ABB RobotStudio station: c.rspag

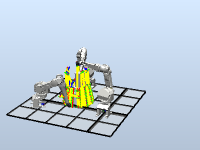
--- station ---
Station c (saved by RobotStudio 6.8.8148.134)
Controller pr3, task T_ROB1: task frame (RAPID world) sits at (2229.65, 1960.18, 0) mm, rotated rx 0 ry 0 rz 180 deg in the station
Controller pr2, task T_ROB1: task frame (RAPID world) sits at (-440.11, 3060.43, 0) mm, rotated rx 0 ry 0 rz -60 deg in the station
Controller pr1
  mechanical unit ROB_1: IRB5510_12A_1100_1500__01, 6 joints, base frame (0, 0, 0) mm
Controller pr2
  mechanical unit ROB_1: IRB5510_12A_1100_1500__01_2, 6 joints, base frame (0, 0, 0) mm
Controller pr3
  mechanical unit ROB_1: IRB5510_12A_1100_1500__01_3, 6 joints, base frame (0, 0, 0) mm
Layout (positions relative to the parent item):
  - IRB5510_12A_1100_1500__01 [mechanism, from Robots\IRB5510_12A_1100_1500__01.rslib] at (0, 0, 0) mm; joint values [1.3542, 0.2117, -0.2881, 5.1047, -1.3259, -6.4536] (rad or m)
  - Workpiece1 [part] at (525.52, 1641.26, 0) mm
  - SmartComponent_1 [smart component]
      signals: DI dipainting
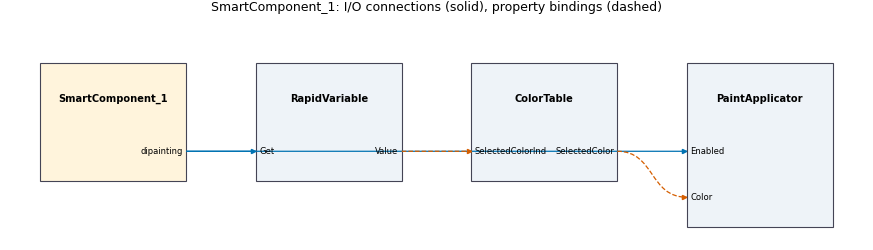
      connections:
        SmartComponent_1.dipainting -> RapidVariable.Get
        SmartComponent_1.dipainting -> PaintApplicator.Enabled
        RapidVariable.Value => ColorTable.SelectedColorIndex
        ColorTable.SelectedColor => PaintApplicator.Color
    - RapidVariable [smart component, from Components\RapidVariable.rslib] at (525.52, 1641.26, 0) mm
        properties: DataType=num; Controller=pr1; Task=T_ROB1; Module=Module1; Variable=ColorIndex; Value=1
    - ColorTable [smart component, from Components\ColorTable.rslib]
        properties: NumColors=2; SelectedColorIndex=1; SelectedColor=-65536; Color0=-8323328; Color1=-65536
    - PaintApplicator [smart component, from Components\PaintApplicator.rslib] at (380.08, 1590.25, 1937.3) mm, rotated rx -165.29 ry -4.8 rz -35.6 deg
        properties: Part=Workpiece1; Color=-65536; ShowPreviewCone=true; Strength=1; Range=0.5; Width=0.1; Height=0.1
  - IRB5510_12A_1100_1500__01_2 [mechanism, from Robots\IRB5510_12A_1100_1500__01.rslib] at (-440.11, 3060.43, 0) mm, rotated rx 0 ry 0 rz -60 deg; joint values [-0.3666, 1.0855, 0.2681, -2.8851, 1.0858, 0.687] (rad or m)
  - SmartComponent_2 [smart component]
      signals: DI dipainting2
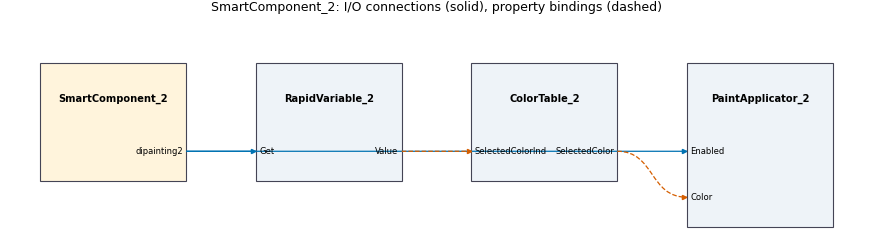
      connections:
        SmartComponent_2.dipainting2 -> RapidVariable_2.Get
        SmartComponent_2.dipainting2 -> PaintApplicator_2.Enabled
        RapidVariable_2.Value => ColorTable_2.SelectedColorIndex
        ColorTable_2.SelectedColor => PaintApplicator_2.Color
    - PaintApplicator_2 [smart component, from Components\PaintApplicator.rslib] at (-112.67, 1718.9, 64) mm, rotated rx -102.66 ry 3.38 rz -125.56 deg
        properties: Part=Workpiece1; Color=-65536; ShowPreviewCone=true; Strength=1; Range=0.5; Width=0.1; Height=0.1
    - RapidVariable_2 [smart component, from Components\RapidVariable.rslib]
        properties: DataType=num; Controller=pr2; Task=T_ROB1; Module=Module1; Variable=ColorIndex2; Value=1
    - ColorTable_2 [smart component, from Components\ColorTable.rslib]
        properties: NumColors=2; SelectedColorIndex=1; SelectedColor=-65536; Color0=-16711936; Color1=-65536
  - IRB5510_12A_1100_1500__01_3 [mechanism, from Robots\IRB5510_12A_1100_1500__01.rslib] at (2229.65, 1960.18, 0) mm, rotated rx 0 ry 0 rz 180 deg; joint values [0.099, 0.1133, 0.783, 6.9211, 0.1129, -9.8516] (rad or m)
  - SmartComponent_3 [smart component]
      signals: DI dipainting3
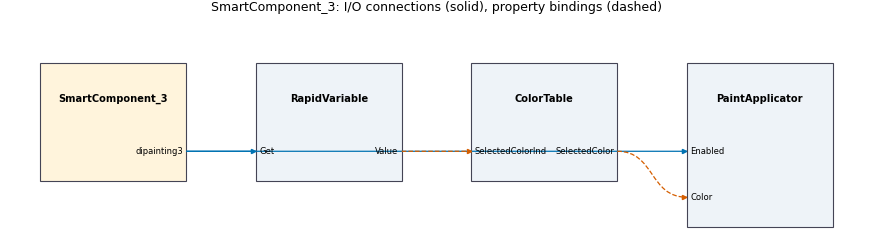
      connections:
        SmartComponent_3.dipainting3 -> RapidVariable.Get
        SmartComponent_3.dipainting3 -> PaintApplicator.Enabled
        RapidVariable.Value => ColorTable.SelectedColorIndex
        ColorTable.SelectedColor => PaintApplicator.Color
    - ColorTable [smart component, from Components\ColorTable.rslib]
        properties: NumColors=2; SelectedColorIndex=1; SelectedColor=-65536; Color0=-16711936; Color1=-65536
    - PaintApplicator [smart component, from Components\PaintApplicator.rslib] at (1182.52, 1870.98, 835.06) mm, rotated rx -177.35 ry -34.28 rz 170.77 deg
        properties: Part=Workpiece1; Color=-65536; ShowPreviewCone=true; Strength=1; Range=0.5; Width=0.1; Height=0.1
    - RapidVariable [smart component, from Components\RapidVariable.rslib]
        properties: DataType=num; Controller=pr3; Task=T_ROB1; Module=Module1; Variable=ColorIndex3; Value=1
Attachment: PaintApplicator is attached to IRB5510_12A_1100_1500__01 / Link6
Attachment: RapidVariable is attached to Workpiece1
Attachment: PaintApplicator_2 is attached to IRB5510_12A_1100_1500__01_2 / Link6
Attachment: PaintApplicator is attached to IRB5510_12A_1100_1500__01_3 / Link6
Station logic (signal -> signal, property => property):
  pr1.do1 -> SmartComponent_1.dipainting
  pr2.do2 -> SmartComponent_2.dipainting2
  pr3.do3 -> SmartComponent_3.dipainting3
Targets, tools, work objects and paths stored in the station and not in the controller backup, written as RAPID:
! task T_ROB1
MODULE Module1
  CONST robtarget Target_20_8_1:=[[1168.457580802,482.978083743,355.510491805],[0.383636594,-0.280466499,0.519275457,-0.710291846],[0,0,0,0],[9E+09,9E+09,9E+09,9E+09,9E+09,9E+09]];
ENDMODULE


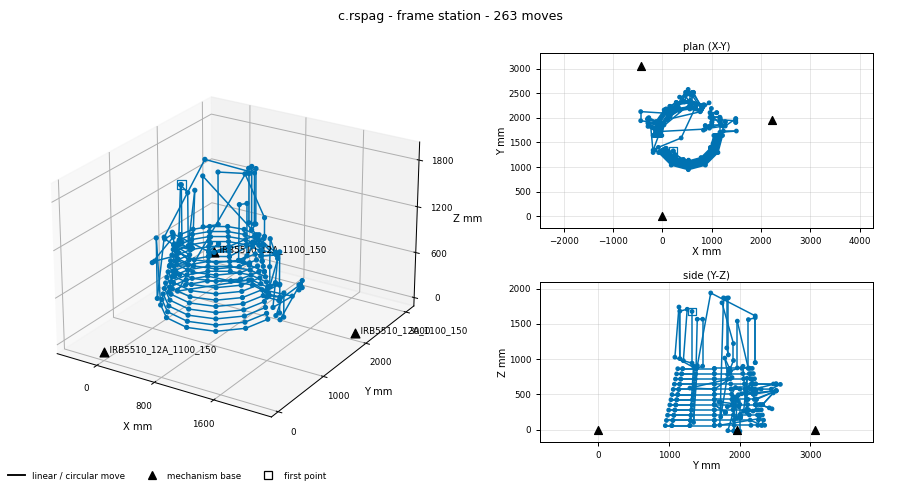
[picture p0: tool path of c.rspag in frame station, 263 of 265 moves have a stored position in this frame; points joined in program order, loops and branches not executed]
--- Backups/pr1/RAPID/TASK0/SYSMOD/userlog.sys ---
module userlog(sysmodule)



   local const num MAX_LOG_SIZE   := 100000; ! Size in bytes.
   local const num MAX_LOG_FILES  := 5;
   local const num MAX_LOG_BUFFER := 20; ! Entries to keep before flushing.



   ! Keep persistent to survive restarts and share between tasks.
   pers string stUserLogBuffer{MAX_LOG_BUFFER};
   pers string stUserLogTime{MAX_LOG_BUFFER};
   pers num nUserLogIndex;
   pers num nUserLogFileNo;

   pers bool bUserBufAddSem;
   pers bool bUserFlushSem;



   proc PntUserLog(string stMessage \Switch Flush)
      BufferAdd stMessage;
      if Present(Flush)
         FlushBuffer;
   endproc



   local proc BufferAdd(string stMessage)
      var bool bTimeOut;

      WaitUntil TestAndSet(bUserBufAddSem) \MaxTime := 1 \TimeFlag := bTimeOut;
      if bTimeOut then
         ErrWrite "PntUserLog Error", "Buffer Add Semaphore Timeout";
         bUserBufAddSem := false; ! Force release.
         return;
      endif

      stUserLogBuffer{nUserLogIndex} := stMessage;
      stUserLogTime{nUserLogIndex} := CDate() + " " + CTime();

      Incr nUserLogIndex;
      if nUserLogIndex > MAX_LOG_BUFFER then
         ! Must be flushed.
         FlushBuffer;
      endif

      bUserBufAddSem := false; ! Release.
   error
      if errno = ERR_OUTOFBND then
         Decr nUserLogIndex;
         retry;
      endif
   endproc



   local proc FlushBuffer()
      var bool bTimeOut;
      var iodev ioLog;
      var string stLogFile;

      WaitUntil TestAndSet(bUserFlushSem) \MaxTime := 1 \TimeFlag := bTimeOut;
      if bTimeOut then
         ErrWrite "PntUserLog Error", "Flush Semaphore Timeout";
         bUserFlushSem := false; ! Force release.
         return;
      endif

      if nUserLogIndex <= 1 then
         bUserFlushSem := false;
         return; ! Buffer empty, nothing to flush.
      endif

      stLogFile := "HOME:/logs/user" + ValToStr(nUserLogFileNo) + ".log";

      Open stLogFile, ioLog \Append;
      for i from 1 to nUserLogIndex - 1 do ! Will normally be incremented to one above.
         Write ioLog, stUserLogTime{i} + " " \NoNewLine;
         Write ioLog, stUserLogBuffer{i};
      endfor
      Close ioLog;
      nUserLogIndex := 1;

      if FileSize(stLogFile) > MAX_LOG_SIZE then
         Incr nUserLogFileNo;
         if nUserLogFileNo > MAX_LOG_FILES
            nUserLogFileNo := 1;

         stLogFile := "HOME:/logs/user" + ValToStr(nUserLogFileNo) + ".log";
         Open stLogFile, ioLog;
         Close ioLog;
      endif

      bUserFlushSem := false;
   error
      nUserLogIndex := 1;
      bUserFlushSem := false;
      return;
   endproc



   proc InitUserLog()
      bUserBufAddSem := false;
      bUserFlushSem := false;
      if nUserLogIndex = 0
         nUserLogIndex := 1;
      if nUserLogFileNo = 0
         nUserLogFileNo := 1;
   endproc



endmodule

--- Backups/pr1/RAPID/TASK1/PROGMOD/Module1.mod ---
MODULE Module1
	CONST robtarget Target_10:=[[220.972076113,1325.461164863,1675.045963445],[0.428514417,-0.848693424,-0.003788423,-0.309968569],[0,-2,0,-1],[9E+09,9E+09,9E+09,9E+09,9E+09,9E+09]];
	CONST robtarget Target_20:=[[220.972027283,1325.461318707,943.383318713],[0.428514341,-0.848693578,-0.003788679,-0.30996825],[0,-3,1,-1],[9E+09,9E+09,9E+09,9E+09,9E+09,9E+09]];
	CONST robtarget Target_30:=[[255.876169889,1202.287029937,977.735293127],[0.428514201,-0.848694161,-0.00378949,-0.309966838],[0,-3,1,-1],[9E+09,9E+09,9E+09,9E+09,9E+09,9E+09]];
	CONST robtarget Target_40:=[[255.876146336,1256.809125064,1706.135963599],[0.428515168,-0.848693816,-0.003790024,-0.30996644],[0,-2,0,-1],[9E+09,9E+09,9E+09,9E+09,9E+09,9E+09]];

    CONST robtarget Target_50:=[[423.854082514,1152.351337183,1679.753004286],[0.470738228,-0.862443821,-0.062003712,-0.175361671],[0,-1,-1,-1],[9E+09,9E+09,9E+09,9E+09,9E+09,9E+09]];
    CONST robtarget Target_60:=[[423.854188981,1152.351291133,1007.412938276],[0.470738104,-0.862443793,-0.062004223,-0.17536196],[0,0,-3,-1],[9E+09,9E+09,9E+09,9E+09,9E+09,9E+09]];
    PERS num ColorIndex:=1;
	CONST robtarget Target_70:=[[530.439659908,1082.627182458,1027.159892696],[0.48639792,-0.862240028,-0.096330933,-0.103341902],[0,0,-2,-1],[9E+09,9E+09,9E+09,9E+09,9E+09,9E+09]];
	CONST robtarget Target_100:=[[76.862753625,1382.222294523,864.109062315],[0.54301355,-0.674637975,0.389502299,-0.313508925],[0,0,0,0],[9E+09,9E+09,9E+09,9E+09,9E+09,9E+09]];
	CONST robtarget Target_110:=[[266.489526282,1192.595596051,864.109062259],[0.605652882,-0.752460843,0.201621223,-0.162284158],[0,0,0,0],[9E+09,9E+09,9E+09,9E+09,9E+09,9E+09]];
	CONST robtarget Target_120:=[[525.524468822,1123.187410427,864.109061963],[0.627017992,-0.779004774,0,0],[0,-2,0,0],[9E+09,9E+09,9E+09,9E+09,9E+09,9E+09]];
	CONST robtarget Target_130:=[[784.559411363,1192.595596051,864.109062259],[0.605652882,-0.752460843,-0.201621223,0.162284158],[0,0,0,0],[9E+09,9E+09,9E+09,9E+09,9E+09,9E+09]];
	CONST robtarget Target_140:=[[974.18618402,1382.222294523,864.109062315],[0.54301355,-0.674637975,-0.389502299,0.313508925],[0,0,0,0],[9E+09,9E+09,9E+09,9E+09,9E+09,9E+09]];
	CONST robtarget Target_150:=[[1043.594471035,1641.25720958,864.109061867],[0.443368761,-0.550839666,-0.55083945,0.443368587],[0,1,1,1],[9E+09,9E+09,9E+09,9E+09,9E+09,9E+09]];
	CONST robtarget Target_150_2:=[[1059.621736679,1641.257203305,790.841560504],[0.443368761,-0.550839666,-0.55083945,0.443368587],[0,1,1,1],[9E+09,9E+09,9E+09,9E+09,9E+09,9E+09]];
	CONST robtarget Target_140_2:=[[988.066201213,1374.208657999,790.841560977],[0.54301355,-0.674637975,-0.389502299,0.313508925],[0,0,0,0],[9E+09,9E+09,9E+09,9E+09,9E+09,9E+09]];
	CONST robtarget Target_130_2:=[[792.573042484,1178.715575754,790.841560918],[0.605652882,-0.752460843,-0.201621223,0.162284158],[0,0,0,0],[9E+09,9E+09,9E+09,9E+09,9E+09,9E+09]];
	CONST robtarget Target_120_2:=[[525.524468822,1107.160144759,790.841560605],[0.627017992,-0.779004774,0,0],[0,-2,0,0],[9E+09,9E+09,9E+09,9E+09,9E+09,9E+09]];
	CONST robtarget Target_110_2:=[[258.475895161,1178.715575754,790.841560918],[0.605652882,-0.752460843,0.201621223,-0.162284158],[0,0,0,0],[9E+09,9E+09,9E+09,9E+09,9E+09,9E+09]];
	CONST robtarget Target_100_2:=[[62.982736432,1374.208657999,790.841560977],[0.54301355,-0.674637975,0.389502299,-0.313508925],[0,0,0,0],[9E+09,9E+09,9E+09,9E+09,9E+09,9E+09]];
	CONST robtarget Target_100_3:=[[49.102719239,1366.195021476,717.574059638],[0.54301355,-0.674637975,0.389502299,-0.313508925],[0,0,0,0],[9E+09,9E+09,9E+09,9E+09,9E+09,9E+09]];
	CONST robtarget Target_110_3:=[[250.462264041,1164.835555457,717.574059576],[0.605652882,-0.752460843,0.201621223,-0.162284158],[0,0,0,0],[9E+09,9E+09,9E+09,9E+09,9E+09,9E+09]];
	CONST robtarget Target_120_3:=[[525.524468822,1091.13287909,717.574059248],[0.627017992,-0.779004774,0,0],[0,-2,0,0],[9E+09,9E+09,9E+09,9E+09,9E+09,9E+09]];
	CONST robtarget Target_130_3:=[[800.586673604,1164.835555457,717.574059576],[0.605652882,-0.752460843,-0.201621223,0.162284158],[0,0,0,0],[9E+09,9E+09,9E+09,9E+09,9E+09,9E+09]];
	CONST robtarget Target_140_3:=[[1001.946218406,1366.195021476,717.574059638],[0.54301355,-0.674637975,-0.389502299,0.313508925],[0,0,0,0],[9E+09,9E+09,9E+09,9E+09,9E+09,9E+09]];
	CONST robtarget Target_150_3:=[[1075.649002323,1641.257197029,717.574059141],[0.443368761,-0.550839666,-0.55083945,0.443368587],[0,1,1,1],[9E+09,9E+09,9E+09,9E+09,9E+09,9E+09]];
	CONST robtarget Target_150_4:=[[1091.676267967,1641.257190755,644.306557778],[0.443368761,-0.550839666,-0.55083945,0.443368587],[0,1,1,1],[9E+09,9E+09,9E+09,9E+09,9E+09,9E+09]];
	CONST robtarget Target_140_4:=[[1015.826235599,1358.181384951,644.306558301],[0.54301355,-0.674637975,-0.389502299,0.313508925],[0,0,0,0],[9E+09,9E+09,9E+09,9E+09,9E+09,9E+09]];
	CONST robtarget Target_130_4:=[[808.600304726,1150.95553516,644.306558236],[0.605652882,-0.752460843,-0.201621223,0.162284158],[0,0,0,0],[9E+09,9E+09,9E+09,9E+09,9E+09,9E+09]];
	CONST robtarget Target_120_4:=[[525.524468822,1075.105613423,644.306557889],[0.627017992,-0.779004774,0,0],[0,-2,0,0],[9E+09,9E+09,9E+09,9E+09,9E+09,9E+09]];
	CONST robtarget Target_110_4:=[[242.448632919,1150.95553516,644.306558236],[0.605652882,-0.752460843,0.201621223,-0.162284158],[0,0,0,0],[9E+09,9E+09,9E+09,9E+09,9E+09,9E+09]];
	CONST robtarget Target_100_4:=[[35.222702046,1358.181384951,644.306558301],[0.54301355,-0.674637975,0.389502299,-0.313508925],[0,0,0,0],[9E+09,9E+09,9E+09,9E+09,9E+09,9E+09]];
	CONST robtarget Target_100_5:=[[21.342684853,1350.167748427,571.039056963],[0.54301355,-0.674637975,0.389502299,-0.313508925],[0,0,0,0],[9E+09,9E+09,9E+09,9E+09,9E+09,9E+09]];
	CONST robtarget Target_110_5:=[[234.435001798,1137.075514863,571.039056895],[0.605652882,-0.752460843,0.201621223,-0.162284158],[0,0,0,0],[9E+09,9E+09,9E+09,9E+09,9E+09,9E+09]];
	CONST robtarget Target_120_5:=[[525.524468822,1059.078347755,571.039056531],[0.627017992,-0.779004774,0,0],[0,-2,0,0],[9E+09,9E+09,9E+09,9E+09,9E+09,9E+09]];
	CONST robtarget Target_130_5:=[[816.613935847,1137.075514863,571.039056895],[0.605652882,-0.752460843,-0.201621223,0.162284158],[0,0,0,0],[9E+09,9E+09,9E+09,9E+09,9E+09,9E+09]];
	CONST robtarget Target_140_5:=[[1029.706252792,1350.167748427,571.039056963],[0.54301355,-0.674637975,-0.389502299,0.313508925],[0,0,0,0],[9E+09,9E+09,9E+09,9E+09,9E+09,9E+09]];
	CONST robtarget Target_150_5:=[[1107.703533611,1641.25718448,571.039056415],[0.443368761,-0.550839666,-0.55083945,0.443368587],[0,1,1,1],[9E+09,9E+09,9E+09,9E+09,9E+09,9E+09]];
	CONST robtarget Target_150_6:=[[1123.730799255,1641.257178205,497.771555052],[0.443368761,-0.550839666,-0.55083945,0.443368587],[0,1,0,1],[9E+09,9E+09,9E+09,9E+09,9E+09,9E+09]];
	CONST robtarget Target_140_6:=[[1043.586269985,1342.154111903,497.771555625],[0.54301355,-0.674637975,-0.389502299,0.313508925],[0,0,0,0],[9E+09,9E+09,9E+09,9E+09,9E+09,9E+09]];
	CONST robtarget Target_130_6:=[[824.627566968,1123.195494566,497.771555554],[0.605652882,-0.752460843,-0.201621223,0.162284158],[0,0,0,0],[9E+09,9E+09,9E+09,9E+09,9E+09,9E+09]];
	CONST robtarget Target_120_6:=[[525.524468822,1043.051082087,497.771555173],[0.627017992,-0.779004774,0,0],[0,-2,0,0],[9E+09,9E+09,9E+09,9E+09,9E+09,9E+09]];
	CONST robtarget Target_110_6:=[[226.421370677,1123.195494566,497.771555554],[0.605652882,-0.752460843,0.201621223,-0.162284158],[0,0,0,0],[9E+09,9E+09,9E+09,9E+09,9E+09,9E+09]];
	CONST robtarget Target_100_6:=[[7.46266766,1342.154111903,497.771555625],[0.54301355,-0.674637975,0.389502299,-0.313508925],[0,0,0,0],[9E+09,9E+09,9E+09,9E+09,9E+09,9E+09]];
	CONST robtarget Target_100_7:=[[-6.417349533,1334.140475379,424.504054287],[0.54301355,-0.674637975,0.389502299,-0.313508925],[0,0,0,0],[9E+09,9E+09,9E+09,9E+09,9E+09,9E+09]];
	CONST robtarget Target_110_7:=[[218.407739556,1109.315474269,424.504054213],[0.605652882,-0.752460843,0.201621223,-0.162284158],[0,-2,0,0],[9E+09,9E+09,9E+09,9E+09,9E+09,9E+09]];
	CONST robtarget Target_120_7:=[[525.524468822,1027.023816419,424.504053815],[0.627017992,-0.779004774,0,0],[0,-2,0,0],[9E+09,9E+09,9E+09,9E+09,9E+09,9E+09]];
	CONST robtarget Target_130_7:=[[832.641198089,1109.315474269,424.504054213],[0.605652882,-0.752460843,-0.201621223,0.162284158],[0,0,0,0],[9E+09,9E+09,9E+09,9E+09,9E+09,9E+09]];
	CONST robtarget Target_140_7:=[[1057.466287178,1334.140475379,424.504054287],[0.54301355,-0.674637975,-0.389502299,0.313508925],[0,0,0,0],[9E+09,9E+09,9E+09,9E+09,9E+09,9E+09]];
	CONST robtarget Target_150_7:=[[1139.758064899,1641.25717193,424.504053689],[0.443368761,-0.550839666,-0.55083945,0.443368587],[0,1,0,1],[9E+09,9E+09,9E+09,9E+09,9E+09,9E+09]];
	CONST robtarget Target_150_8:=[[1155.785330543,1641.257165655,351.236552326],[0.443368761,-0.550839666,-0.55083945,0.443368587],[0,1,0,1],[9E+09,9E+09,9E+09,9E+09,9E+09,9E+09]];
	CONST robtarget Target_140_8:=[[1071.346304371,1326.126838855,351.236552949],[0.54301355,-0.674637975,-0.389502299,0.313508925],[0,0,0,0],[9E+09,9E+09,9E+09,9E+09,9E+09,9E+09]];
	CONST robtarget Target_130_8:=[[840.65482921,1095.435453972,351.236552872],[0.605652882,-0.752460843,-0.201621223,0.162284158],[0,0,0,0],[9E+09,9E+09,9E+09,9E+09,9E+09,9E+09]];
	CONST robtarget Target_120_8:=[[525.524468822,1010.996550751,351.236552457],[0.627017992,-0.779004774,0,0],[0,-2,0,0],[9E+09,9E+09,9E+09,9E+09,9E+09,9E+09]];
	CONST robtarget Target_110_8:=[[210.394108435,1095.435453972,351.236552872],[0.605652882,-0.752460843,0.201621223,-0.162284158],[0,-2,0,0],[9E+09,9E+09,9E+09,9E+09,9E+09,9E+09]];
	CONST robtarget Target_100_8:=[[-20.297366726,1326.126838855,351.236552949],[0.54301355,-0.674637975,0.389502299,-0.313508925],[0,0,0,0],[9E+09,9E+09,9E+09,9E+09,9E+09,9E+09]];
	CONST robtarget Target_100_9:=[[-34.177383919,1318.113202331,277.969051611],[0.54301355,-0.674637975,0.389502299,-0.313508925],[0,0,0,0],[9E+09,9E+09,9E+09,9E+09,9E+09,9E+09]];
	CONST robtarget Target_110_9:=[[202.380477314,1081.555433675,277.969051531],[0.605652882,-0.752460843,0.201621223,-0.162284158],[0,-2,0,0],[9E+09,9E+09,9E+09,9E+09,9E+09,9E+09]];
	CONST robtarget Target_120_9:=[[525.524468822,994.969285083,277.969051099],[0.627017992,-0.779004774,0,0],[0,-2,0,0],[9E+09,9E+09,9E+09,9E+09,9E+09,9E+09]];
	CONST robtarget Target_130_9:=[[848.668460331,1081.555433675,277.969051531],[0.605652882,-0.752460843,-0.201621223,0.162284158],[0,0,0,0],[9E+09,9E+09,9E+09,9E+09,9E+09,9E+09]];
	CONST robtarget Target_140_9:=[[1085.226321564,1318.113202331,277.969051611],[0.54301355,-0.674637975,-0.389502299,0.313508925],[0,0,0,0],[9E+09,9E+09,9E+09,9E+09,9E+09,9E+09]];
	CONST robtarget Target_150_9:=[[1171.812596187,1641.25715938,277.969050963],[0.443368761,-0.550839666,-0.55083945,0.443368587],[0,1,0,1],[9E+09,9E+09,9E+09,9E+09,9E+09,9E+09]];
	CONST robtarget Target_150_10:=[[1187.839861831,1641.257153105,204.7015496],[0.443368761,-0.550839666,-0.55083945,0.443368587],[0,1,0,1],[9E+09,9E+09,9E+09,9E+09,9E+09,9E+09]];
	CONST robtarget Target_140_10:=[[1099.106338757,1310.099565807,204.701550273],[0.54301355,-0.674637975,-0.389502299,0.313508925],[0,0,0,0],[9E+09,9E+09,9E+09,9E+09,9E+09,9E+09]];
	CONST robtarget Target_130_10:=[[856.682091452,1067.675413378,204.70155019],[0.605652882,-0.752460843,-0.201621223,0.162284158],[0,0,0,0],[9E+09,9E+09,9E+09,9E+09,9E+09,9E+09]];
	CONST robtarget Target_120_10:=[[525.524468822,978.942019415,204.701549741],[0.627017992,-0.779004774,0,0],[0,-2,0,0],[9E+09,9E+09,9E+09,9E+09,9E+09,9E+09]];
	CONST robtarget Target_110_10:=[[194.366846193,1067.675413378,204.70155019],[0.605652882,-0.752460843,0.201621223,-0.162284158],[0,-2,0,0],[9E+09,9E+09,9E+09,9E+09,9E+09,9E+09]];
	CONST robtarget Target_100_10:=[[-48.057401112,1310.099565807,204.701550273],[0.54301355,-0.674637975,0.389502299,-0.313508925],[0,0,0,0],[9E+09,9E+09,9E+09,9E+09,9E+09,9E+09]];
	CONST robtarget Target_100_11:=[[-61.937418307,1302.085929287,131.43404893],[0.54301355,-0.674637975,0.389502299,-0.313508925],[0,0,0,0],[9E+09,9E+09,9E+09,9E+09,9E+09,9E+09]];
	CONST robtarget Target_110_11:=[[186.353215075,1053.795393083,131.434048844],[0.605652882,-0.752460843,0.201621223,-0.162284158],[0,-2,0,0],[9E+09,9E+09,9E+09,9E+09,9E+09,9E+09]];
	CONST robtarget Target_120_11:=[[525.524468822,962.914753743,131.434048386],[0.627017992,-0.779004774,0,0],[0,-2,0,0],[9E+09,9E+09,9E+09,9E+09,9E+09,9E+09]];
	CONST robtarget Target_130_11:=[[864.69572257,1053.795393083,131.434048844],[0.605652882,-0.752460843,-0.201621223,0.162284158],[0,0,0,0],[9E+09,9E+09,9E+09,9E+09,9E+09,9E+09]];
	CONST robtarget Target_140_11:=[[1112.986355952,1302.085929287,131.43404893],[0.54301355,-0.674637975,-0.389502299,0.313508925],[0,0,0,0],[9E+09,9E+09,9E+09,9E+09,9E+09,9E+09]];
	CONST robtarget Target_150_11:=[[1203.867127477,1641.257146827,131.434048238],[0.443368761,-0.550839666,-0.55083945,0.443368587],[0,1,0,1],[9E+09,9E+09,9E+09,9E+09,9E+09,9E+09]];
	CONST robtarget Target_150_12:=[[1219.894393122,1641.257140552,58.166546875],[0.443368761,-0.550839666,-0.55083945,0.443368587],[0,1,0,1],[9E+09,9E+09,9E+09,9E+09,9E+09,9E+09]];
	CONST robtarget Target_140_12:=[[1126.866373146,1294.072292764,58.166547592],[0.54301355,-0.674637975,-0.389502299,0.313508925],[0,0,0,0],[9E+09,9E+09,9E+09,9E+09,9E+09,9E+09]];
	CONST robtarget Target_130_12:=[[872.70935369,1039.915372786,58.166547503],[0.605652882,-0.752460843,-0.201621223,0.162284158],[0,0,0,0],[9E+09,9E+09,9E+09,9E+09,9E+09,9E+09]];
	CONST robtarget Target_120_12:=[[525.524468822,946.887488074,58.166547029],[0.627017992,-0.779004774,0,0],[0,-2,0,0],[9E+09,9E+09,9E+09,9E+09,9E+09,9E+09]];
	CONST robtarget Target_110_12:=[[178.339583955,1039.915372786,58.166547503],[0.605652882,-0.752460843,0.201621223,-0.162284158],[0,-2,0,0],[9E+09,9E+09,9E+09,9E+09,9E+09,9E+09]];
	CONST robtarget Target_100_12:=[[-75.817435501,1294.072292764,58.166547592],[0.54301355,-0.674637975,0.389502299,-0.313508925],[0,0,0,0],[9E+09,9E+09,9E+09,9E+09,9E+09,9E+09]];
	CONST robtarget Target_80:=[[530.440073821,1140.249250209,1737.815045101],[0.48639809,-0.862239917,-0.096330687,-0.103342255],[0,-1,-1,-1],[9E+09,9E+09,9E+09,9E+09,9E+09,9E+09]];
    CONST robtarget Target_140_13:=[[974.187304287,1399.238179155,1565.111954946],[0.543014556,-0.674640793,-0.389500166,0.313503768],[0,1,1,1],[9E+09,9E+09,9E+09,9E+09,9E+09,9E+09]];
    CONST robtarget Target_140_14:=[[1030.490260811,1475.545352143,1565.111998843],[0.515440165,-0.640382182,-0.443579682,0.357028239],[0,1,1,1],[9E+09,9E+09,9E+09,9E+09,9E+09,9E+09]];
    CONST robtarget Target_140_15:=[[1030.490207729,1475.545264413,900.097554314],[0.515440526,-0.640382753,-0.443579297,0.357027171],[0,1,1,1],[9E+09,9E+09,9E+09,9E+09,9E+09,9E+09]];
    CONST robtarget Target_170:=[[-159.590405899,1346.881037064,899.74471457],[0.53978193,-0.670632312,0.396368893,-0.319028949],[1,2,-3,-1],[9E+09,9E+09,9E+09,9E+09,9E+09,9E+09]];
    CONST robtarget Target_160:=[[-159.590245756,1346.880552292,103.379449569],[0.539782978,-0.670632306,0.396367617,-0.319028775],[1,2,-3,-1],[9E+09,9E+09,9E+09,9E+09,9E+09,9E+09]];
	CONST robtarget Target_180:=[[-81.501829709,1400.411105396,907.726080868],[0.539781583,-0.670633815,0.396368094,-0.31902737],[1,2,-3,-1],[9E+09,9E+09,9E+09,9E+09,9E+09,9E+09]];
	CONST robtarget Target_190:=[[380.07970095,1590.248446999,1937.301071362],[0.109074939,-0.945100203,0.297835821,-0.078626254],[0,3,-5,-1],[9E+09,9E+09,9E+09,9E+09,9E+09,9E+09]];
PROC Path_10()
	    ColorIndex:=1;
        Set do1;
        WaitTime 1;
        MoveL Target_10,v1000,z100,tool0\WObj:=wobj0;
	    MoveL Target_20,v1000,z100,tool0\WObj:=wobj0;
	    MoveL Target_30,v1000,z100,tool0\WObj:=wobj0;
	    MoveL Target_40,v1000,z100,tool0\WObj:=wobj0;
        MoveL Target_50,v1000,z100,tool0\WObj:=wobj0;
        MoveL Target_60,v1000,z100,tool0\WObj:=wobj0;
        MoveL Target_80,v1000,z100,tool0\WObj:=wobj0;
        MoveL Target_70,v1000,z100,tool0\WObj:=wobj0;
        MoveL Target_100,v1000,z100,tool0\WObj:=wobj0;
        MoveL Target_110,v1000,z100,tool0\WObj:=wobj0;
        MoveL Target_120,v1000,z100,tool0\WObj:=wobj0;
        MoveL Target_130,v1000,z100,tool0\WObj:=wobj0;
        MoveL Target_140,v1000,z100,tool0\WObj:=wobj0;
        MoveL Target_140_13,v1000,z100,tool0\WObj:=wobj0;
        MoveL Target_140_14,v1000,z100,tool0\WObj:=wobj0;
        MoveL Target_140_15,v1000,z100,tool0\WObj:=wobj0;
        MoveL Target_140,v1000,z100,tool0\WObj:=wobj0;
        MoveL Target_150,v1000,z100,tool0\WObj:=wobj0;
        MoveL Target_150_2,v1000,z100,tool0\WObj:=wobj0;
        MoveL Target_140_2,v1000,z100,tool0\WObj:=wobj0;
        MoveL Target_130_2,v1000,z100,tool0\WObj:=wobj0;
        MoveL Target_120_2,v1000,z100,tool0\WObj:=wobj0;
        MoveL Target_110_2,v1000,z100,tool0\WObj:=wobj0;
        MoveL Target_100_2,v1000,z100,tool0\WObj:=wobj0;
        MoveL Target_100_3,v1000,z100,tool0\WObj:=wobj0;
        MoveL Target_110_3,v1000,z100,tool0\WObj:=wobj0;
        MoveL Target_120_3,v1000,z100,tool0\WObj:=wobj0;
        MoveL Target_130_3,v1000,z100,tool0\WObj:=wobj0;
        MoveL Target_140_3,v1000,z100,tool0\WObj:=wobj0;
        MoveL Target_150_3,v1000,z100,tool0\WObj:=wobj0;
        MoveL Target_150_4,v1000,z100,tool0\WObj:=wobj0;
        MoveL Target_140_4,v1000,z100,tool0\WObj:=wobj0;
        MoveL Target_130_4,v1000,z100,tool0\WObj:=wobj0;
        MoveL Target_120_4,v1000,z100,tool0\WObj:=wobj0;
        MoveL Target_110_4,v1000,z100,tool0\WObj:=wobj0;
        MoveL Target_100_4,v1000,z100,tool0\WObj:=wobj0;
        MoveL Target_100_5,v1000,z100,tool0\WObj:=wobj0;
        MoveL Target_110_5,v1000,z100,tool0\WObj:=wobj0;
        MoveL Target_120_5,v1000,z100,tool0\WObj:=wobj0;
        MoveL Target_130_5,v1000,z100,tool0\WObj:=wobj0;
        MoveL Target_140_5,v1000,z100,tool0\WObj:=wobj0;
        MoveL Target_150_5,v1000,z100,tool0\WObj:=wobj0;
        MoveL Target_150_6,v1000,z100,tool0\WObj:=wobj0;
        MoveL Target_140_6,v1000,z100,tool0\WObj:=wobj0;
        MoveL Target_130_6,v1000,z100,tool0\WObj:=wobj0;
        MoveL Target_120_6,v1000,z100,tool0\WObj:=wobj0;
        MoveL Target_110_6,v1000,z100,tool0\WObj:=wobj0;
        MoveL Target_100_6,v1000,z100,tool0\WObj:=wobj0;
        MoveL Target_100_7,v1000,z100,tool0\WObj:=wobj0;
        MoveL Target_110_7,v1000,z100,tool0\WObj:=wobj0;
        MoveL Target_120_7,v1000,z100,tool0\WObj:=wobj0;
        MoveL Target_130_7,v1000,z100,tool0\WObj:=wobj0;
        MoveL Target_140_7,v1000,z100,tool0\WObj:=wobj0;
        MoveL Target_150_7,v1000,z100,tool0\WObj:=wobj0;
        MoveL Target_150_8,v1000,z100,tool0\WObj:=wobj0;
        MoveL Target_140_8,v1000,z100,tool0\WObj:=wobj0;
        MoveL Target_130_8,v1000,z100,tool0\WObj:=wobj0;
        MoveL Target_120_8,v1000,z100,tool0\WObj:=wobj0;
        MoveL Target_110_8,v1000,z100,tool0\WObj:=wobj0;
        MoveL Target_100_8,v1000,z100,tool0\WObj:=wobj0;
        MoveL Target_100_9,v1000,z100,tool0\WObj:=wobj0;
        MoveL Target_110_9,v1000,z100,tool0\WObj:=wobj0;
        MoveL Target_120_9,v1000,z100,tool0\WObj:=wobj0;
        MoveL Target_130_9,v1000,z100,tool0\WObj:=wobj0;
        MoveL Target_140_9,v1000,z100,tool0\WObj:=wobj0;
        MoveL Target_150_9,v1000,z100,tool0\WObj:=wobj0;
        MoveL Target_150_10,v1000,z100,tool0\WObj:=wobj0;
        MoveL Target_140_10,v1000,z100,tool0\WObj:=wobj0;
        MoveL Target_130_10,v1000,z100,tool0\WObj:=wobj0;
        MoveL Target_120_10,v1000,z100,tool0\WObj:=wobj0;
        MoveL Target_110_10,v1000,z100,tool0\WObj:=wobj0;
        MoveL Target_100_10,v1000,z100,tool0\WObj:=wobj0;
        MoveL Target_100_11,v1000,z100,tool0\WObj:=wobj0;
		MoveL Target_110_11,v1000,z100,tool0\WObj:=wobj0;
		MoveL Target_120_11,v1000,z100,tool0\WObj:=wobj0;
		MoveL Target_130_11,v1000,z100,tool0\WObj:=wobj0;
		MoveL Target_140_11,v1000,z100,tool0\WObj:=wobj0;
		MoveL Target_150_11,v1000,z100,tool0\WObj:=wobj0;
		MoveL Target_150_12,v1000,z100,tool0\WObj:=wobj0;
		MoveL Target_140_12,v1000,z100,tool0\WObj:=wobj0;
		MoveL Target_130_12,v1000,z100,tool0\WObj:=wobj0;
		MoveL Target_120_12,v1000,z100,tool0\WObj:=wobj0;
		MoveL Target_110_12,v1000,z100,tool0\WObj:=wobj0;
		MoveL Target_100_12,v1000,z100,tool0\WObj:=wobj0;
        MoveL Target_170,v1000,z100,tool0\WObj:=wobj0;
        MoveL Target_160,v1000,z100,tool0\WObj:=wobj0;
		MoveL Target_180,v1000,z100,tool0\WObj:=wobj0;
		MoveL Target_190,v1000,z100,tool0\WObj:=wobj0;
        WaitTime 1;
        Reset do1;
    ENDPROC

ENDMODULE

--- Backups/pr1/RAPID/TASK1/SYSMOD/custmain.sys ---
module custmain(sysmodule)



   proc InitCustMain()
      !
      ! Insert RAPID code for start at main here...
      !
   endproc



   proc PreMainCustom()
      !
      ! This will be executed before a paint program...
      !
   endproc



   proc PostMainCustom()
      !
      ! This will be executed after a paint program...
      !
   endproc



endmodule

--- Backups/pr1/RAPID/TASK1/SYSMOD/robdata.sys ---
module robdata(sysmodule)

   ! Note: This file can be used to add custom tools/speeds/zones.
   ! Uncomment any standard tools here, if they are needed.



   ! Default generic gun (10x5cm, 60 degree):
   pers tooldata tDefGun_Tip := [true,[[50,0,100],[0.866025,0,0.5,0]],[2,[0,0,50],[1,0,0,0],0,0,0]];
   pers tooldata tDefGun_100 := [true,[[136.6,0,150],[0.866025,0,0.5,0]],[2,[0,0,50],[1,0,0,0],0,0,0]];
   pers tooldata tDefGun_200 := [true,[[223.2,0,200],[0.866025,0,0.5,0]],[2,[0,0,50],[1,0,0,0],0,0,0]];

   ! Robobel 925:
   !pers tooldata tRB925_200 := [true,[[290.1,0,540],[0.866025,0,0.5,0]],[8,[0,0,33],[1,0,0,0],0,0,0]];
   !pers tooldata tRB925_250 := [true,[[333.4,0,565],[0.866025,0,0.5,0]],[8,[0,0,33],[1,0,0,0],0,0,0]];

   ! HCEBELL:
   !pers tooldata tHCEBELL_0   := [true,[[142.9,0,427.5],[0.866025,0,0.5,0]],[10,[0,-40,250],[1,0,0,0],0,0,0]];
   !pers tooldata tHCEBELL_150 := [true,[[272.8,0,502.5],[0.866025,0,0.5,0]],[11,[0,40,250],[1,0,0,0],0,0,0]];
   !pers tooldata tHCEBELL_200 := [true,[[316.1,0,527.5],[0.866025,0,0.5,0]],[11,[0,40,250],[1,0,0,0],0,0,0]];
   !pers tooldata tHCEBELL_250 := [true,[[359.4,0,552.5],[0.866025,0,0.5,0]],[11,[0,40,250],[1,0,0,0],0,0,0]];
   !pers tooldata tHCEBELL_300 := [true,[[402.7,0,577.5],[0.866025,0,0.5,0]],[11,[0,40,250],[1,0,0,0],0,0,0]];

   ! ABB Ecco Gun:
   !pers tooldata tEccoGun_Tip := [true,[[1.8,0,156.6],[0.965926,0,0.258819,0]],[2,[0,0,120],[1,0,0,0],0,0,0]];
   !pers tooldata tEccoGun_200 := [true,[[101.8,0,329.8],[0.965926,0,0.258819,0]],[2,[0,0,120],[1,0,0,0],0,0,0]];
   !pers tooldata tEccoGun_250 := [true,[[126.8,0,373.1],[0.965926,0,0.258819,0]],[2,[0,0,120],[1,0,0,0],0,0,0]];
   !pers tooldata tEccoGun_300 := [true,[[151.8,0,416.4],[0.965926,0,0.258819,0]],[2,[0,0,120],[1,0,0,0],0,0,0]];

   ! G1Direct (short bracket):
   !pers tooldata tG1Direct_300 := [true,[[571.58,0,450],[0.866025,0,0.5,0]],[6.6,[135.2,0,174.1],[1,0,0,0],0,0,0]];
   !pers tooldata tG1Direct_250 := [true,[[528.28,0,425],[0.866025,0,0.5,0]],[6.6,[135.2,0,174.1],[1,0,0,0],0,0,0]];
   !pers tooldata tG1Direct_200 := [true,[[484.97,0,400],[0.866025,0,0.5,0]],[6.6,[135.2,0,174.1],[1,0,0,0],0,0,0]];

   ! G1_Long Braket:
   !pers tooldata tG1V3_200L := [true,[[487,0,502.3],[0.866025,0,0.5,0]],[8,[140.6,0,170],[1,0,0,0],0,0,0]];
   !pers tooldata tG1V3_250L := [true,[[524,0,528.9],[0.866025,0,0.5,0]],[8,[140.6,0,170],[1,0,0,0],0,0,0]];
   !pers tooldata tG1V3_300L := [true,[[549,0,571.6],[0.866025,0,0.5,0]],[8,[140.6,0,170],[1,0,0,0],0,0,0]];

   ! Cartridge Bell:
   !pers tooldata tCBS_0   := [true,[[121.25,0,415],[0.866025,0,0.5,0]],[5.5,[30,0,225],[1,0,0,0],0,0,0]];
   !pers tooldata tCBS_100 := [true,[[207.85,0,465],[0.866025,0,0.5,0]],[5.5,[30,0,225],[1,0,0,0],0,0,0]];
   !pers tooldata tCBS_200 := [true,[[294.45,0,515],[0.866025,0,0.5,0]],[5.5,[30,0,225],[1,0,0,0],0,0,0]];
   !pers tooldata tCBS_250 := [true,[[337.75,0,540],[0.866025,0,0.5,0]],[5.5,[30,0,225],[1,0,0,0],0,0,0]];
   !pers tooldata tCBS_300 := [true,[[381.05,0,565],[0.866025,0,0.5,0]],[5.5,[30,0,225],[1,0,0,0],0,0,0]];

   ! Cartridge Gun:
   !pers tooldata tCGS_0   := [true,[[127.44,0,418.5],[0.866025,0,0.5,0]],[8.1,[30,0,225],[1,0,0,0],0,0,0]];
   !pers tooldata tCGS_100 := [true,[[214.04,0,468.5],[0.866025,0,0.5,0]],[8.1,[30,0,225],[1,0,0,0],0,0,0]];
   !pers tooldata tCGS_200 := [true,[[300.64,0,518.5],[0.866025,0,0.5,0]],[8.1,[30,0,225],[1,0,0,0],0,0,0]];
   !pers tooldata tCGS_250 := [true,[[343.95,0,543.5],[0.866025,0,0.5,0]],[8.1,[30,0,225],[1,0,0,0],0,0,0]];
   !pers tooldata tCGS_300 := [true,[[387.11,0,568.5],[0.866025,0,0.5,0]],[8.1,[30,0,225],[1,0,0,0],0,0,0]];

   ! Robobel 926:
   !pers tooldata tRB926TD_0   := [true,[[116.9,0,470],[0.866025,0,0.5,0]],[5.5,[30,0,225],[1,0,0,0],0,0,0]];
   !pers tooldata tRB926TD_100 := [true,[[203.5,0,520],[0.866025,0,0.5,0]],[5.5,[30,0,225],[1,0,0,0],0,0,0]];
   !pers tooldata tRB926TD_120 := [true,[[220.8,0,530],[0.866025,0,0.5,0]],[5.5,[30,0,225],[1,0,0,0],0,0,0]];
   !pers tooldata tRB926TD_150 := [true,[[246.8,0,545],[0.866025,0,0.5,0]],[5.5,[30,0,225],[1,0,0,0],0,0,0]];
   !pers tooldata tRB926TD_200 := [true,[[290.1,0,570],[0.866025,0,0.5,0]],[5.5,[30,0,225],[1,0,0,0],0,0,0]];
   !pers tooldata tRB926TD_250 := [true,[[333.4,0,595],[0.866025,0,0.5,0]],[5.5,[30,0,225],[1,0,0,0],0,0,0]];
   !pers tooldata tRB926TD_300 := [true,[[376.7,0,620],[0.866025,0,0.5,0]],[5.5,[30,0,225],[1,0,0,0],0,0,0]];

   ! Robobel 625TD:
   !pers tooldata tRB625TD_0   := [true,[[116.9,0,420],[0.866025,0,0.5,0]],[5.1,[30,0,215],[1,0,0,0],0,0,0]];
   !pers tooldata tRB625TD_150 := [true,[[246.8,0,495],[0.866025,0,0.5,0]],[5.1,[30,0,215],[1,0,0,0],0,0,0]];
   !pers tooldata tRB625TD_200 := [true,[[290.1,0,520],[0.866025,0,0.5,0]],[5.1,[30,0,215],[1,0,0,0],0,0,0]];
   !pers tooldata tRB625TD_250 := [true,[[333.4,0,545],[0.866025,0,0.5,0]],[5.1,[30,0,215],[1,0,0,0],0,0,0]];
   !pers tooldata tRB625TD_300 := [true,[[376.7,0,570],[0.866025,0,0.5,0]],[5.1,[30,0,215],[1,0,0,0],0,0,0]];

   ! Robobel 951TD:
   !pers tooldata tRB951TD_0   := [true,[[116.9,0,470],[0.866025,0,0.5,0]],[6.3,[30,0,220],[1,0,0,0],0,0,0]];
   !pers tooldata tRB951TD_100 := [true,[[203.5,0,520],[0.866025,0,0.5,0]],[6.3,[30,0,220],[1,0,0,0],0,0,0]];
   !pers tooldata tRB951TD_120 := [true,[[220.8,0,530],[0.866025,0,0.5,0]],[6.3,[30,0,220],[1,0,0,0],0,0,0]];
   !pers tooldata tRB951TD_150 := [true,[[246.8,0,545],[0.866025,0,0.5,0]],[6.3,[30,0,220],[1,0,0,0],0,0,0]];
   !pers tooldata tRB951TD_200 := [true,[[290.1,0,570],[0.866025,0,0.5,0]],[6.3,[30,0,220],[1,0,0,0],0,0,0]];
   !pers tooldata tRB951TD_250 := [true,[[333.4,0,595],[0.866025,0,0.5,0]],[6.3,[30,0,220],[1,0,0,0],0,0,0]];
   !pers tooldata tRB951TD_300 := [true,[[376.7,0,620],[0.866025,0,0.5,0]],[6.3,[30,0,220],[1,0,0,0],0,0,0]];

   ! Robobel 951CBS /40pai/50pai/70pai:
   !pers tooldata tRB951CBS_0   := [true,[[121.25,0,415],[0.866025,0,0.5,0]],[6.3,[55,0,225],[1,0,0,0],0,0,0]];
   !pers tooldata tRB951CBS_100 := [true,[[207.85,0,465],[0.866025,0,0.5,0]],[6.3,[55,0,225],[1,0,0,0],0,0,0]];
   !pers tooldata tRB951CBS_120 := [true,[[225.17,0,475],[0.866025,0,0.5,0]],[6.3,[55,0,225],[1,0,0,0],0,0,0]];
   !pers tooldata tRB951CBS_150 := [true,[[251.15,0,490],[0.866025,0,0.5,0]],[6.3,[55,0,225],[1,0,0,0],0,0,0]];
   !pers tooldata tRB951CBS_200 := [true,[[294.45,0,515],[0.866025,0,0.5,0]],[6.3,[55,0,225],[1,0,0,0],0,0,0]];
   !pers tooldata tRB951CBS_250 := [true,[[337.75,0,540],[0.866025,0,0.5,0]],[6.3,[55,0,225],[1,0,0,0],0,0,0]];
   !pers tooldata tRB951CBS_300 := [true,[[381.05,0,565],[0.866025,0,0.5,0]],[6.3,[55,0,225],[1,0,0,0],0,0,0]];

   ! Interior Robobel951CBS /30pai:
   !pers tooldata tInteriorCBS_0   := [true,[[99.6,0,402.5],[0.866025,0,0.5,0]],[6.3,[30,0,220],[1,0,0,0],0,0,0]];
   !pers tooldata tInteriorCBS_100 := [true,[[186.2,0,452.5],[0.866025,0,0.5,0]],[6.3,[30,0,220],[1,0,0,0],0,0,0]];
   !pers tooldata tInteriorCBS_120 := [true,[[246.8,0,487.5],[0.866025,0,0.5,0]],[6.3,[30,0,220],[1,0,0,0],0,0,0]];
   !pers tooldata tInteriorCBS_150 := [true,[[272.8,0,502.5],[0.866025,0,0.5,0]],[6.3,[30,0,220],[1,0,0,0],0,0,0]];
   !pers tooldata tInteriorCBS_200 := [true,[[316.1,0,527.5],[0.866025,0,0.5,0]],[6.3,[30,0,220],[1,0,0,0],0,0,0]];
   !pers tooldata tInteriorCBS_250 := [true,[[359.4,0,552.5],[0.866025,0,0.5,0]],[6.3,[30,0,220],[1,0,0,0],0,0,0]];
   !pers tooldata tInteriorCBS_300 := [true,[[402.7,0,577.5],[0.866025,0,0.5,0]],[6.3,[30,0,220],[1,0,0,0],0,0,0]];

   ! Interior Robobel951 /30pai:
   !pers tooldata tInterior951_0   := [true,[[138.6,0,482.5],[0.866025,0,0.5,0]],[6.3,[30,0,220],[1,0,0,0],0,0,0]];
   !pers tooldata tInterior951_100 := [true,[[225.17,0,532.5],[0.866025,0,0.5,0]],[6.3,[30,0,220],[1,0,0,0],0,0,0]];
   !pers tooldata tInterior951_120 := [true,[[242.49,0,542.5],[0.866025,0,0.5,0]],[6.3,[30,0,220],[1,0,0,0],0,0,0]];
   !pers tooldata tInterior951_150 := [true,[[268.47,0,557.5],[0.866025,0,0.5,0]],[6.3,[30,0,220],[1,0,0,0],0,0,0]];
   !pers tooldata tInterior951_200 := [true,[[311.77,0,582.5],[0.866025,0,0.5,0]],[6.3,[30,0,220],[1,0,0,0],0,0,0]];
   !pers tooldata tInterior951_250 := [true,[[355.07,0,607.5],[0.866025,0,0.5,0]],[6.3,[30,0,220],[1,0,0,0],0,0,0]];
   !pers tooldata tInterior951_300 := [true,[[398.37,0,632.5],[0.866025,0,0.5,0]],[6.3,[30,0,220],[1,0,0,0],0,0,0]];

   ! RB-1000WSC (700cc Cartridge):
   !pers tooldata tRB1000WSC_0     := [true,[[121.25,0,450],[0.866025,0,0.5,0]],[13.0,[-52,0,270],[1,0,0,0],0,0,0]];
   !pers tooldata tRB1000WSC_100   := [true,[[207.85,0,500],[0.866025,0,0.5,0]],[13.0,[-52,0,270],[1,0,0,0],0,0,0]];
   !pers tooldata tRB1000WSC_150   := [true,[[251.15,0,525],[0.866025,0,0.5,0]],[13.0,[-52,0,270],[1,0,0,0],0,0,0]];
   !pers tooldata tRB1000WSC_200   := [true,[[294.45,0,550],[0.866025,0,0.5,0]],[13.0,[-52,0,270],[1,0,0,0],0,0,0]];
   !pers tooldata tRB1000WSC_250   := [true,[[337.75,0,575],[0.866025,0,0.5,0]],[13.0,[-52,0,270],[1,0,0,0],0,0,0]];
   !pers tooldata tRB1000WSC_300   := [true,[[381.05,0,600],[0.866025,0,0.5,0]],[13.0,[-52,0,270],[1,0,0,0],0,0,0]];
   !pers tooldata tRB1000WSC_teach := [true,[[-259.801,0,230],[0.866025,0,0.5,0]],[13.0,[-52,0,270],[1,0,0,0],0,0,0]];

   ! RB-1000SAD (Robobel Type):
   !pers tooldata tRB1000SAD_0   := [true,[[181.9,0,472.5],[0.866025,0,0.5,0]],[10.7,[31,0,260],[1,0,0,0],0,0,0]];
   !pers tooldata tRB1000SAD_100 := [true,[[268.5,0,522.5],[0.866025,0,0.5,0]],[10.7,[31,0,260],[1,0,0,0],0,0,0]];
   !pers tooldata tRB1000SAD_150 := [true,[[311.8,0,547.5],[0.866025,0,0.5,0]],[10.7,[31,0,260],[1,0,0,0],0,0,0]];
   !pers tooldata tRB1000SAD_200 := [true,[[355.1,0,572.5],[0.866025,0,0.5,0]],[10.7,[31,0,260],[1,0,0,0],0,0,0]];
   !pers tooldata tRB1000SAD_250 := [true,[[398.4,0,597.5],[0.866025,0,0.5,0]],[10.7,[31,0,260],[1,0,0,0],0,0,0]];
   !pers tooldata tRB1000SAD_300 := [true,[[441.7,0,622.5],[0.866025,0,0.5,0]],[10.7,[31,0,260],[1,0,0,0],0,0,0]];

   ! RB-1000SSD (Robobel Type):
   !pers tooldata tRB1000SSD_0   := [true,[[181.9,0,472.5],[0.866025,0,0.5,0]],[10.7,[31,0,260],[1,0,0,0],0,0,0]];
   !pers tooldata tRB1000SSD_100 := [true,[[268.5,0,522.5],[0.866025,0,0.5,0]],[10.7,[31,0,260],[1,0,0,0],0,0,0]];
   !pers tooldata tRB1000SSD_150 := [true,[[311.8,0,547.5],[0.866025,0,0.5,0]],[10.7,[31,0,260],[1,0,0,0],0,0,0]];
   !pers tooldata tRB1000SSD_200 := [true,[[355.1,0,572.5],[0.866025,0,0.5,0]],[10.7,[31,0,260],[1,0,0,0],0,0,0]];
   !pers tooldata tRB1000SSD_250 := [true,[[398.4,0,597.5],[0.866025,0,0.5,0]],[10.7,[31,0,260],[1,0,0,0],0,0,0]];
   !pers tooldata tRB1000SSD_300 := [true,[[441.7,0,622.5],[0.866025,0,0.5,0]],[10.7,[31,0,260],[1,0,0,0],0,0,0]];

   ! RoboBel021-mini for HollowWrist
   !pers tooldata tRB1021min_tip := [true,[[170.0,0,200],[0.866025,0,0.5,0]],[2.8,[80,0,140],[1,0,0,0],0,0,0]];
   !pers tooldata tRB1021min_100 := [true,[[256.6,0,250],[0.866025,0,0.5,0]],[2.8,[80,0,140],[1,0,0,0],0,0,0]];
   !pers tooldata tRB1021min_150 := [true,[[299.9,0,275],[0.866025,0,0.5,0]],[2.8,[80,0,140],[1,0,0,0],0,0,0]];
   !pers tooldata tRB1021min_200 := [true,[[343.2,0,300],[0.866025,0,0.5,0]],[2.8,[80,0,140],[1,0,0,0],0,0,0]];
   !pers tooldata tRB1021min_250 := [true,[[386.5,0,325],[0.866025,0,0.5,0]],[2.8,[80,0,140],[1,0,0,0],0,0,0]];
   !pers tooldata tRB1021min_300 := [true,[[429.8,0,350],[0.866025,0,0.5,0]],[2.8,[80,0,140],[1,0,0,0],0,0,0]];
   !pers tooldata tRB1021min_350 := [true,[[473.1,0,375],[0.866025,0,0.5,0]],[2.8,[80,0,140],[1,0,0,0],0,0,0]];
   !pers tooldata tRB1021min_400 := [true,[[516.4,0,400],[0.866025,0,0.5,0]],[2.8,[80,0,140],[1,0,0,0],0,0,0]];

   ! AGMD PRO gun with single attachment for Hollow wrist. No Dump (3HNM 10123-1)
   !pers tooldata tAGP10123_TIP:=[TRUE,[[ 52,0,198],[0.866025,0,0.5,0]],[1.490,[0, 0, 101],[1,0,0,0],0,0,0]];
   !pers tooldata tAGP10123_150:=[TRUE,[[178,0,273],[0.866025,0,0.5,0]],[1.490,[0, 0, 101],[1,0,0,0],0,0,0]];
   !pers tooldata tAGP10123_225:=[TRUE,[[243,0,310],[0.866025,0,0.5,0]],[1.490,[0, 0, 101],[1,0,0,0],0,0,0]];
   !pers tooldata tAGP10123_300:=[TRUE,[[308,0,348],[0.866025,0,0.5,0]],[1.490,[0, 0, 101],[1,0,0,0],0,0,0]];

   ! AGMD PRO gun with single attachment for Hollow wrist. With Dump. (3HNM 10121-1)
   !pers tooldata tAGP10121_TIP:=[TRUE,[[ 52,0,198],[0.866025,0,0.5,0]],[1.510,[0, 0, 100],[1,0,0,0],0,0,0]];
   !pers tooldata tAGP10121_150:=[TRUE,[[178,0,273],[0.866025,0,0.5,0]],[1.510,[0, 0, 100],[1,0,0,0],0,0,0]];
   !pers tooldata tAGP10121_225:=[TRUE,[[243,0,310],[0.866025,0,0.5,0]],[1.510,[0, 0, 100],[1,0,0,0],0,0,0]];
   !pers tooldata tAGP10121_300:=[TRUE,[[308,0,348],[0.866025,0,0.5,0]],[1.510,[0, 0, 100],[1,0,0,0],0,0,0]];

   ! AGMD PRO gun with single attachment for Hollow wirst. With Dump, MPAC version. (3HNA 017776-001)
   !pers tooldata tAGP17776_TIP:=[TRUE,[[ 52,0,198],[0.866025,0,0.5,0]],[1.520,[0,0,103],[1,0,0,0],0,0,0]];
   !pers tooldata tAGP17776_150:=[TRUE,[[178,0,273],[0.866025,0,0.5,0]],[1.520,[0,0,103],[1,0,0,0],0,0,0]];
   !pers tooldata tAGP17776_225:=[TRUE,[[243,0,310],[0.866025,0,0.5,0]],[1.520,[0,0,103],[1,0,0,0],0,0,0]];
   !pers tooldata tAGP17776_300:=[TRUE,[[308,0,348],[0.866025,0,0.5,0]],[1.520,[0,0,103],[1,0,0,0],0,0,0]];

   ! RB1000-EXT Short Bracket
   !pers tooldata RB1000EXTS_TIP:=[TRUE,[[362.5,0,121.0],[0.866025,0,0.5,0]],[10.2,[130, 0, 182],[1,0,0,0],0,0,0]];
   !pers tooldata RB1000EXTS_100:=[TRUE,[[400.5,0,352.2],[0.866025,0,0.5,0]],[10.2,[130, 0, 182],[1,0,0,0],0,0,0]];
   !pers tooldata RB1000EXTS_200:=[TRUE,[[487.1,0,402.2],[0.866025,0,0.5,0]],[10.2,[130, 0, 182],[1,0,0,0],0,0,0]];
   !pers tooldata RB1000EXTS_250:=[TRUE,[[530.4,0,427.2],[0.866025,0,0.5,0]],[10.2,[130, 0, 182],[1,0,0,0],0,0,0]];
   !pers tooldata RB1000EXTS_300:=[TRUE,[[573.7,0,452.2],[0.866025,0,0.5,0]],[10.2,[130, 0, 182],[1,0,0,0],0,0,0]];

   ! RB1000-EXT Long Bracket
   !pers tooldata RB1000EXTL_TIP:=[TRUE,[[362.5,0,221.0],[0.866025,0,0.5,0]],[10.6,[130, 0, 260],[1,0,0,0],0,0,0]];
   !pers tooldata RB1000EXTL_100:=[TRUE,[[400.5,0,452.2],[0.866025,0,0.5,0]],[10.6,[130, 0, 260],[1,0,0,0],0,0,0]];
   !pers tooldata RB1000EXTL_200:=[TRUE,[[487.1,0,502.2],[0.866025,0,0.5,0]],[10.6,[130, 0, 260],[1,0,0,0],0,0,0]];
   !pers tooldata RB1000EXTL_250:=[TRUE,[[530.4,0,527.2],[0.866025,0,0.5,0]],[10.6,[130, 0, 260],[1,0,0,0],0,0,0]];
   !pers tooldata RB1000EXTL_300:=[TRUE,[[573.7,0,552.2],[0.866025,0,0.5,0]],[10.6,[130, 0, 260],[1,0,0,0],0,0,0]];

   ! RB1000i-SSD
   !pers tooldata RB1000iSSD_TIP:=[TRUE,[[228.6,0,480.0],[0.866025,0,0.5,0]],[9.0,[52, 0, 293],[1,0,0,0],0,0,0]];
   !pers tooldata RB1000iSSD_100:=[TRUE,[[315.2,0,530.0],[0.866025,0,0.5,0]],[9.0,[52, 0, 293],[1,0,0,0],0,0,0]];
   !pers tooldata RB1000iSSD_200:=[TRUE,[[401.8,0,580.0],[0.866025,0,0.5,0]],[9.0,[52, 0, 293],[1,0,0,0],0,0,0]];
   !pers tooldata RB1000iSSD_250:=[TRUE,[[445.1,0,605.0],[0.866025,0,0.5,0]],[9.0,[52, 0, 293],[1,0,0,0],0,0,0]];
   !pers tooldata RB1000iSSD_300:=[TRUE,[[488.4,0,630.0],[0.866025,0,0.5,0]],[9.0,[52, 0, 293],[1,0,0,0],0,0,0]];

   ! RB1000i-SAD
   !pers tooldata RB1000iSAD_TIP:=[TRUE,[[228.6,0,480.0],[0.866025,0,0.5,0]],[9.0,[52, 0, 293],[1,0,0,0],0,0,0]];
   !pers tooldata RB1000iSAD_100:=[TRUE,[[315.2,0,530.0],[0.866025,0,0.5,0]],[9.0,[52, 0, 293],[1,0,0,0],0,0,0]];
   !pers tooldata RB1000iSAD_200:=[TRUE,[[401.8,0,580.0],[0.866025,0,0.5,0]],[9.0,[52, 0, 293],[1,0,0,0],0,0,0]];
   !pers tooldata RB1000iSAD_250:=[TRUE,[[445.1,0,605.0],[0.866025,0,0.5,0]],[9.0,[52, 0, 293],[1,0,0,0],0,0,0]];
   !pers tooldata RB1000iSAD_300:=[TRUE,[[488.4,0,630.0],[0.866025,0,0.5,0]],[9.0,[52, 0, 293],[1,0,0,0],0,0,0]];

   ! RB1000i-S2K
   !pers tooldata RB1000iS2K_TIP:=[TRUE,[[228.6,0,480.0],[0.866025,0,0.5,0]],[9.0,[52, 0, 293],[1,0,0,0],0,0,0]];
   !pers tooldata RB1000iS2K_100:=[TRUE,[[315.2,0,530.0],[0.866025,0,0.5,0]],[9.0,[52, 0, 293],[1,0,0,0],0,0,0]];
   !pers tooldata RB1000iS2K_200:=[TRUE,[[401.8,0,580.0],[0.866025,0,0.5,0]],[9.0,[52, 0, 293],[1,0,0,0],0,0,0]];
   !pers tooldata RB1000iS2K_250:=[TRUE,[[445.1,0,605.0],[0.866025,0,0.5,0]],[9.0,[52, 0, 293],[1,0,0,0],0,0,0]];
   !pers tooldata RB1000iS2K_300:=[TRUE,[[488.4,0,630.0],[0.866025,0,0.5,0]],[9.0,[52, 0, 293],[1,0,0,0],0,0,0]];

   ! RB1000i External charge, Long Bracket
   !pers tooldata RB1000iEXTL_TIP:=[TRUE,[[313.9,0,402.3],[0.866025,0,0.5,0]],[11.3,[128.5, 0, 266],[1,0,0,0],0,0,0]];
   !pers tooldata RB1000iEXTL_100:=[TRUE,[[400.5,0,452.3],[0.866025,0,0.5,0]],[11.3,[128.5, 0, 266],[1,0,0,0],0,0,0]];
   !pers tooldata RB1000iEXTL_200:=[TRUE,[[487.1,0,502.3],[0.866025,0,0.5,0]],[11.3,[128.5, 0, 266],[1,0,0,0],0,0,0]];
   !pers tooldata RB1000iEXTL_250:=[TRUE,[[530.4,0,527.3],[0.866025,0,0.5,0]],[11.3,[128.5, 0, 266],[1,0,0,0],0,0,0]];
   !pers tooldata RB1000iEXTL_300:=[TRUE,[[573.7,0,552.3],[0.866025,0,0.5,0]],[11.3,[128.5, 0, 266],[1,0,0,0],0,0,0]];

   ! RB1000i External charge, Short Bracket
   !pers tooldata RB1000iEXTS_TIP:=[TRUE,[[313.9,0,302.3],[0.866025,0,0.5,0]],[10.8,[136.6, 0, 188.4],[1,0,0,0],0,0,0]];
   !pers tooldata RB1000iEXTS_100:=[TRUE,[[400.5,0,352.3],[0.866025,0,0.5,0]],[10.8,[136.6, 0, 188.4],[1,0,0,0],0,0,0]];
   !pers tooldata RB1000iEXTS_200:=[TRUE,[[487.1,0,402.3],[0.866025,0,0.5,0]],[10.8,[136.6, 0, 188.4],[1,0,0,0],0,0,0]];
   !pers tooldata RB1000iEXTS_250:=[TRUE,[[530.4,0,427.3],[0.866025,0,0.5,0]],[10.8,[136.6, 0, 188.4],[1,0,0,0],0,0,0]];
   !pers tooldata RB1000iEXTS_300:=[TRUE,[[573.7,0,452.3],[0.866025,0,0.5,0]],[10.8,[136.6, 0, 188.4],[1,0,0,0],0,0,0]];

   ! RB1000-CE (Compact External)
   !pers tooldata RB1000CE_TIP:=[TRUE,[[233.8,0,370.0],[0.866025,0,0.5,0]],[9.5,[72, 0, 236],[1,0,0,0],0,0,0]];
   !pers tooldata RB1000CE_100:=[TRUE,[[320.4,0,420.0],[0.866025,0,0.5,0]],[9.5,[72, 0, 236],[1,0,0,0],0,0,0]];
   !pers tooldata RB1000CE_200:=[TRUE,[[407.0,0,470.0],[0.866025,0,0.5,0]],[9.5,[72, 0, 236],[1,0,0,0],0,0,0]];
   !pers tooldata RB1000CE_250:=[TRUE,[[450.3,0,495.0],[0.866025,0,0.5,0]],[9.5,[72, 0, 236],[1,0,0,0],0,0,0]];
   !pers tooldata RB1000CE_300:=[TRUE,[[493.6,0,520.0],[0.866025,0,0.5,0]],[9.5,[72, 0, 236],[1,0,0,0],0,0,0]];



   ! Speed data:
   !const speeddata vPaint50   := [50,300,1000,50];
   !const speeddata vPaint100  := [100,300,100,100];
   !const speeddata vPaint150  := [150,300,150,150];
   !const speeddata vPaint200  := [200,300,200,200];
   !const speeddata vPaint250  := [250,300,250,250];
   !const speeddata vPaint300  := [300,300,300,300];
   !const speeddata vPaint350  := [350,300,350,350];
   !const speeddata vPaint400  := [400,300,400,400];
   !const speeddata vPaint450  := [450,300,450,450];
   !const speeddata vPaint500  := [500,300,500,500];
   !const speeddata vPaint550  := [550,300,1000,500];
   !const speeddata vPaint600  := [600,300,1000,500];
   !const speeddata vPaint650  := [650,300,1000,500];
   !const speeddata vPaint700  := [700,300,1000,500];
   !const speeddata vPaint750  := [750,300,1000,500];
   !const speeddata vPaint800  := [800,300,1000,500];
   !const speeddata vPaint850  := [850,300,1000,500];
   !const speeddata vPaint900  := [900,300,1000,500];
   !const speeddata vPaint950  := [950,300,1000,500];
   !const speeddata vPaint1000 := [1000,300,1000,500];
   !const speeddata vPaint1100 := [1100,300,1000,500];
   !const speeddata vPaint1200 := [1200,300,1000,500];
   !const speeddata vPaint1300 := [1300,300,1000,500];
   !const speeddata vPaint1400 := [1400,300,1000,500];
   !const speeddata vPaint1500 := [1500,300,1000,500];
   !const speeddata vPaint1600 := [1600,300,1000,500];
   !const speeddata vPaint1700 := [1700,300,1000,500];
   !const speeddata vPaint1800 := [1800,300,1000,500];
   !const speeddata vPaint1900 := [1900,300,1000,500];
   !const speeddata vPaint2000 := [2000,300,1000,500];
   !const speeddata vPaint2100 := [2100,300,1000,500];
   !const speeddata vPaint2200 := [2200,300,1000,500];
   !const speeddata vPaint2300 := [2300,300,1000,500];
   !const speeddata vPaint2400 := [2400,300,1000,500];
   !const speeddata vPaint2500 := [2500,300,1000,500];



   ! Speed data (High Flow Bell):
   const speeddata vHFB50   := [50,150,50,50];
   const speeddata vHFB100  := [100,150,100,100];
   const speeddata vHFB150  := [150,150,150,150];
   const speeddata vHFB200  := [200,150,200,200];
   const speeddata vHFB250  := [250,150,250,250];
   const speeddata vHFB300  := [300,150,300,300];
   const speeddata vHFB350  := [350,150,350,350];
   const speeddata vHFB400  := [400,150,400,400];
   const speeddata vHFB450  := [450,150,450,450];
   const speeddata vHFB500  := [500,150,500,500];
   const speeddata vHFB550  := [550,150,1000,500];
   const speeddata vHFB600  := [600,150,1000,500];
   const speeddata vHFB650  := [650,150,1000,500];
   const speeddata vHFB700  := [700,150,1000,500];
   const speeddata vHFB750  := [750,150,1000,500];
   const speeddata vHFB800  := [800,150,1000,500];
   const speeddata vHFB850  := [850,150,1000,500];
   const speeddata vHFB900  := [900,150,1000,500];
   const speeddata vHFB950  := [950,150,1000,500];
   const speeddata vHFB1000 := [1000,150,1000,500];
   const speeddata vHFB1100 := [1100,150,1000,500];
   const speeddata vHFB1200 := [1200,150,1000,500];
   const speeddata vHFB1300 := [1300,150,1000,500];
   const speeddata vHFB1400 := [1400,150,1000,500];
   const speeddata vHFB1500 := [1500,150,1000,500];
   const speeddata vHFB1600 := [1600,150,1000,500];
   const speeddata vHFB1700 := [1700,150,1000,500];
   const speeddata vHFB1800 := [1800,150,1000,500];
   const speeddata vHFB1900 := [1900,150,1000,500];
   const speeddata vHFB2000 := [2000,150,1000,500];
   const speeddata vHFB2100 := [2100,150,1000,500];
   const speeddata vHFB2200 := [2200,150,1000,500];
   const speeddata vHFB2300 := [2300,150,1000,500];
   const speeddata vHFB2400 := [2400,150,1000,500];
   const speeddata vHFB2500 := [2500,150,1000,500];



   ! Zone data:
   !const zonedata zPaint1   := [false,1,1,1,0.15,1,0.15];
   !const zonedata zPaint5   := [false,5,8,8,0.8,8,0.8];
   !const zonedata zPaint10  := [false,10,15,15,1.5,15,1.5];
   !const zonedata zPaint15  := [false,15,23,23,2.3,23,2.3];
   !const zonedata zPaint20  := [false,20,30,30,3,30,3];
   !const zonedata zPaint30  := [false,30,45,45,4.5,45,4.5];
   !const zonedata zPaint40  := [false,40,60,60,6,60,6];
   !const zonedata zPaint50  := [false,50,75,75,7.5,75,7.5];
   !const zonedata zPaint60  := [false,60,90,90,9,90,9];
   !const zonedata zPaint80  := [false,80,120,120,12,120,12];
   !const zonedata zPaint100 := [false,100,150,150,15,150,15];
   !const zonedata zPaint150 := [false,150,225,225,23,225,23];
   !const zonedata zPaint200 := [false,200,300,300,30,300,30];
   !const zonedata zPaint250 := [false,250,375,375,37.5,375,37.5];
   !const zonedata zPaint300 := [false,300,450,450,45,450,45];



endmodule

--- Backups/pr1/RAPID/TASK1/SYSMOD/sysdata.sys ---
module sysdata(sysmodule)

   ! Note: This file is used to store system positions and setup world zones.



   pers tooldata tUserTool0 := [TRUE,[[0,0,0],[1,0,0,0]],[0.001,[0,0,0.001],[1,0,0,0],0,0,0]];

   pers robtarget pHomePos   := [[0,0,0],[9E+09,9E+09,9E+09,9E+09],[-1,-1,1,0],[9E+09,9E+09,9E+09,9E+09,9E+09,9E+09]];
   pers robtarget pMtrlChPos := [[0,0,0],[9E+09,9E+09,9E+09,9E+09],[-1,-1,1,0],[9E+09,9E+09,9E+09,9E+09,9E+09,9E+09]];
   pers robtarget pReadyPos  := [[0,0,0],[9E+09,9E+09,9E+09,9E+09],[-1,-1,1,0],[9E+09,9E+09,9E+09,9E+09,9E+09,9E+09]];
   pers robtarget pUserPos   := [[0,0,0],[9E+09,9E+09,9E+09,9E+09],[-1,-1,1,0],[9E+09,9E+09,9E+09,9E+09,9E+09,9E+09]];

   pers jointtarget jHomePos   := [[9E+09,9E+09,9E+09,9E+09,9E+09,9E+09],[9E+09,9E+09,9E+09,9E+09,9E+09,0]];
   pers jointtarget jMtrlChPos := [[9E+09,9E+09,9E+09,9E+09,9E+09,9E+09],[9E+09,9E+09,9E+09,9E+09,9E+09,0]];
   pers jointtarget jReadyPos  := [[9E+09,9E+09,9E+09,9E+09,9E+09,9E+09],[9E+09,9E+09,9E+09,9E+09,9E+09,0]];
   pers jointtarget jUserPos   := [[9E+09,9E+09,9E+09,9E+09,9E+09,9E+09],[9E+09,9E+09,9E+09,9E+09,9E+09,0]];

   local var wzstationary wzHomePos;
   local var wzstationary wzMtrlChPos;
   local var wzstationary wzReadyPos;
   local var wzstationary wzUserPos;

   local var pos psHomePos   := [0,0,0];
   local var pos psMtrlChPos := [0,0,0];
   local var pos psReadyPos  := [0,0,0];
   local var pos psUserPos   := [0,0,0];

   local var signaldo doHomePosAlias;
   local var signaldo doMtrlChPosAlias;
   local var signaldo doReadyPosAlias;
   local var signaldo doUserPosAlias;



   proc PowerOnWZones()
      var shapedata volHomePos;
      var shapedata volMtrlChPos;
      var shapedata volReadyPos;
      var shapedata volUserPos;

      ! AliasIO requires variables to work.
      var string stHomePos       := "doHomePos";
      var string stMtrlChangePos := "doMtrlChangePos";
      var string stReadyPos      := "doReadyPos";
      var string stUserPos       := "doUserPos";

      psHomePos   := pHomePos.trans;
      psMtrlChPos := pMtrlChPos.trans;
      psReadyPos  := pReadyPos.trans;
      psUserPos   := pUserPos.trans;

      WZSphDef \Inside, volHomePos, psHomePos, 6;
      WZSphDef \Inside, volMtrlChPos, psMtrlChPos, 6;
      WZSphDef \Inside, volReadyPos, psReadyPos, 6;
      WZSphDef \Inside, volUserPos, psUserPos, 6;

      if GetSignal("doHomePos") <> -1000000 then
         AliasIO stHomePos, doHomePosAlias;
         WZDOSet \Stat, wzHomePos \Inside, volHomePos, doHomePosAlias, 1;
      endif
      if GetSignal("doMtrlChangePos") <> -1000000 then
         AliasIO stMtrlChangePos, doMtrlChPosAlias;
         WZDOSet \Stat, wzMtrlChPos \Inside, volMtrlChPos, doMtrlChPosAlias, 1;
      endif
      if GetSignal("doReadyPos") <> -1000000 then
         AliasIO stReadyPos, doReadyPosAlias;
         WZDOSet \Stat, wzReadyPos \Inside, volReadyPos, doReadyPosAlias, 1;
      endif
      if GetSignal("doUserPos") <> -1000000 then
         AliasIO stUserPos, doUserPosAlias;
         WZDOSet \Stat, wzUserPos \Inside, volUserPos, doUserPosAlias, 1;
      endif
   endproc



   proc ConfSettingsOff()
      ConfJ \Off;
      ConfL \Off;
   endproc



endmodule

--- Backups/pr1/RAPID/TASK2/SYSMOD/custcmd.sys ---
module custcmd(sysmodule)



   proc InitCustCmd()
      !
      ! Insert RAPID code for startup here...
      !
   endproc



   proc Cmd1001(num nInParam{*}, inout num nResult, inout num nOutData{*})
      !
      ! Insert RAPID code for command here...
      !
      ErrWrite "Cmd1001",
         ValToStr(nInParam{1}) + "," +
         ValToStr(nInParam{2}) + "," +
         ValToStr(nInParam{3}) + "," +
         ValToStr(nInParam{4}) + "," +
         ValToStr(nInParam{5}) + "," +
         ValToStr(nInParam{6}) + "," +
         ValToStr(nInParam{7}) + "," +
         ValToStr(nInParam{8}) + "," +
         ValToStr(nInParam{9}) + "," +
         ValToStr(nInParam{10});

      nResult := CMD_OK;
   endproc



   proc Cmd1002(num nInParam{*}, inout num nResult, inout num nOutData{*})
      !
      ! Insert RAPID code for command here...
      !
      ErrWrite "Cmd1002", "";

      nOutData{1}  := nInParam{1};
      nOutData{2}  := nInParam{2};
      nOutData{3}  := nInParam{3};
      nOutData{4}  := nInParam{4};
      nOutData{5}  := nInParam{5};
      nOutData{6}  := nInParam{6};
      nOutData{7}  := nInParam{7};
      nOutData{8}  := nInParam{8};
      nOutData{9}  := nInParam{9};
      nOutData{10} := nInParam{10};

      nResult := CMD_OK;
   endproc



endmodule

--- Backups/pr2/RAPID/TASK1/PROGMOD/Module1.mod ---
MODULE Module1
	CONST robtarget Target_10:=[[1415.646117144,575.318702107,868.383001798],[0.180363377,-0.224082776,0.746079989,-0.600516954],[0,-1,-1,0],[9E+09,9E+09,9E+09,9E+09,9E+09,9E+09]];
	CONST robtarget Target_20:=[[1262.279053715,421.461252556,868.38300101],[0.297974422,-0.370202292,0.685418633,-0.55169086],[0,0,0,0],[9E+09,9E+09,9E+09,9E+09,9E+09,9E+09]];
	CONST robtarget Target_30:=[[1182.323114803,219.469621071,868.383000844],[0.403294899,-0.501052053,0.596485774,-0.480109139],[0,0,0,0],[9E+09,9E+09,9E+09,9E+09,9E+09,9E+09]];
	CONST robtarget Target_40:=[[1188.834059745,2.326399704,868.383001217],[0.491980647,-0.611234891,0.482949633,-0.388724329],[-1,-2,0,0],[9E+09,9E+09,9E+09,9E+09,9E+09,9E+09]];
	PERS  num ColorIndex2:=1;
    CONST robtarget Target_10_2:=[[1406.815255754,588.693646744,795.115500523],[0.180363377,-0.224082776,0.746079989,-0.600516954],[0,0,0,0],[9E+09,9E+09,9E+09,9E+09,9E+09,9E+09]];
    CONST robtarget Target_10_3:=[[1397.984394364,602.068591381,721.847999248],[0.180363377,-0.224082776,0.746079989,-0.600516954],[0,0,0,0],[9E+09,9E+09,9E+09,9E+09,9E+09,9E+09]];
    CONST robtarget Target_10_4:=[[1389.153532974,615.443536018,648.580497973],[0.180363377,-0.224082776,0.746079989,-0.600516954],[0,0,0,0],[9E+09,9E+09,9E+09,9E+09,9E+09,9E+09]];
    CONST robtarget Target_10_5:=[[1380.322671584,628.818480655,575.312996698],[0.180363377,-0.224082776,0.746079989,-0.600516954],[0,0,0,0],[9E+09,9E+09,9E+09,9E+09,9E+09,9E+09]];
    CONST robtarget Target_10_6:=[[1371.491810194,642.193425292,502.045495423],[0.180363377,-0.224082776,0.746079989,-0.600516954],[0,0,0,0],[9E+09,9E+09,9E+09,9E+09,9E+09,9E+09]];
    CONST robtarget Target_10_7:=[[1362.660948804,655.568369929,428.777994148],[0.180363377,-0.224082776,0.746079989,-0.600516954],[0,0,0,0],[9E+09,9E+09,9E+09,9E+09,9E+09,9E+09]];
    CONST robtarget Target_10_8:=[[1353.830087414,668.943314566,355.510492873],[0.180363377,-0.224082776,0.746079989,-0.600516954],[0,0,0,0],[9E+09,9E+09,9E+09,9E+09,9E+09,9E+09]];
    CONST robtarget Target_10_9:=[[1344.999226024,682.318259203,282.242991598],[0.180363377,-0.224082776,0.746079989,-0.600516954],[0,0,0,0],[9E+09,9E+09,9E+09,9E+09,9E+09,9E+09]];
    CONST robtarget Target_10_10:=[[1336.168364634,695.69320384,208.975490323],[0.180363377,-0.224082776,0.746079989,-0.600516954],[0,0,0,0],[9E+09,9E+09,9E+09,9E+09,9E+09,9E+09]];
    CONST robtarget Target_20_2:=[[1248.875986156,430.249371297,795.115499695],[0.297974422,-0.370202292,0.685418633,-0.55169086],[0,0,0,0],[9E+09,9E+09,9E+09,9E+09,9E+09,9E+09]];
    CONST robtarget Target_20_3:=[[1235.472918597,439.037490038,721.84799838],[0.297974422,-0.370202292,0.685418633,-0.55169086],[0,0,0,0],[9E+09,9E+09,9E+09,9E+09,9E+09,9E+09]];
    CONST robtarget Target_20_6:=[[1004.561958261,653.663933732,554.541508989],[0.29797094,-0.370202538,0.685421819,-0.551688617],[0,-1,0,0],[9E+09,9E+09,9E+09,9E+09,9E+09,9E+09]];
    CONST robtarget Target_20_7:=[[992.65646245,630.379826759,549.432772181],[0.29797139,-0.370202078,0.68542123,-0.551689415],[0,-1,0,0],[9E+09,9E+09,9E+09,9E+09,9E+09,9E+09]];
    CONST robtarget Target_20_8:=[[1168.457580802,482.978083743,355.510491805],[0.297974423,-0.370202292,0.685418632,-0.55169086],[0,0,0,0],[9E+09,9E+09,9E+09,9E+09,9E+09,9E+09]];
    CONST robtarget Target_20_9:=[[1155.054513243,491.766202484,282.24299049],[0.297974422,-0.370202292,0.685418633,-0.55169086],[0,0,0,0],[9E+09,9E+09,9E+09,9E+09,9E+09,9E+09]];
    CONST robtarget Target_20_10:=[[1141.651445684,500.554321225,208.975489175],[0.297974422,-0.370202292,0.685418633,-0.55169086],[0,0,0,0],[9E+09,9E+09,9E+09,9E+09,9E+09,9E+09]];
    CONST robtarget Target_30_2:=[[1166.536386553,222.235929246,795.11549952],[0.403294899,-0.501052053,0.596485774,-0.480109139],[0,0,0,0],[9E+09,9E+09,9E+09,9E+09,9E+09,9E+09]];
    CONST robtarget Target_30_3:=[[1150.749658303,225.002237421,721.847998196],[0.403294899,-0.501052053,0.596485774,-0.480109139],[0,0,0,0],[9E+09,9E+09,9E+09,9E+09,9E+09,9E+09]];
    CONST robtarget Target_30_4:=[[1134.962930053,227.768545596,648.580496872],[0.403294899,-0.501052053,0.596485774,-0.480109139],[0,0,0,0],[9E+09,9E+09,9E+09,9E+09,9E+09,9E+09]];
    CONST robtarget Target_30_5:=[[1119.176201803,230.534853771,575.312995548],[0.403294899,-0.501052053,0.596485774,-0.480109139],[0,0,0,0],[9E+09,9E+09,9E+09,9E+09,9E+09,9E+09]];
    CONST robtarget Target_30_6:=[[1103.389473553,233.301161946,502.045494224],[0.403294899,-0.501052053,0.596485774,-0.480109139],[0,0,0,0],[9E+09,9E+09,9E+09,9E+09,9E+09,9E+09]];
    CONST robtarget Target_30_7:=[[1087.602745303,236.067470121,428.7779929],[0.403294899,-0.501052054,0.596485774,-0.480109139],[0,0,0,0],[9E+09,9E+09,9E+09,9E+09,9E+09,9E+09]];
    CONST robtarget Target_30_8:=[[1071.816017053,238.833778296,355.510491576],[0.403294899,-0.501052053,0.596485774,-0.480109139],[0,0,0,0],[9E+09,9E+09,9E+09,9E+09,9E+09,9E+09]];
    CONST robtarget Target_30_9:=[[1056.029288803,241.600086471,282.242990252],[0.403294899,-0.501052053,0.596485774,-0.480109139],[0,-2,0,0],[9E+09,9E+09,9E+09,9E+09,9E+09,9E+09]];
    CONST robtarget Target_30_10:=[[1040.242560553,244.366394646,208.975488928],[0.403294899,-0.501052053,0.596485774,-0.480109139],[0,-2,0,0],[9E+09,9E+09,9E+09,9E+09,9E+09,9E+09]];
    CONST robtarget Target_40_2:=[[1173.241436852,-1.380804616,795.115499912],[0.491980647,-0.611234891,0.482949633,-0.388724329],[-1,-2,0,0],[9E+09,9E+09,9E+09,9E+09,9E+09,9E+09]];
    CONST robtarget Target_40_3:=[[1157.648813959,-5.088008936,721.847998607],[0.491980647,-0.611234891,0.482949633,-0.388724329],[-1,-2,0,0],[9E+09,9E+09,9E+09,9E+09,9E+09,9E+09]];
    CONST robtarget Target_40_4:=[[1142.056191066,-8.795213256,648.580497302],[0.491980647,-0.611234891,0.482949633,-0.388724329],[-1,-2,0,0],[9E+09,9E+09,9E+09,9E+09,9E+09,9E+09]];
    CONST robtarget Target_40_5:=[[1126.463568173,-12.502417576,575.312995997],[0.491980647,-0.611234891,0.482949633,-0.388724329],[-1,-2,0,0],[9E+09,9E+09,9E+09,9E+09,9E+09,9E+09]];
    CONST robtarget Target_40_6:=[[1110.87094528,-16.209621896,502.045494692],[0.491980647,-0.611234891,0.482949633,-0.388724329],[-1,-2,0,0],[9E+09,9E+09,9E+09,9E+09,9E+09,9E+09]];
    CONST robtarget Target_40_7:=[[1095.278322387,-19.916826216,428.777993387],[0.491980647,-0.611234891,0.482949633,-0.388724329],[-1,-2,0,0],[9E+09,9E+09,9E+09,9E+09,9E+09,9E+09]];
    CONST robtarget Target_40_8:=[[1079.685699494,-23.624030536,355.510492082],[0.491980647,-0.611234891,0.482949633,-0.388724329],[-1,-2,0,0],[9E+09,9E+09,9E+09,9E+09,9E+09,9E+09]];
    CONST robtarget Target_40_9:=[[1064.093076601,-27.331234856,282.242990777],[0.491980647,-0.611234891,0.482949633,-0.388724329],[-1,-2,0,0],[9E+09,9E+09,9E+09,9E+09,9E+09,9E+09]];
    CONST robtarget Target_40_10:=[[1048.500453708,-31.038439176,208.975489472],[0.491980647,-0.611234891,0.482949633,-0.388724329],[-1,-2,0,0],[9E+09,9E+09,9E+09,9E+09,9E+09,9E+09]];
    CONST robtarget Target_50:=[[1280.748736327,-194.51176644,868.383000926],[0.560373641,-0.696206087,0.349493238,-0.281305783],[-1,-2,0,0],[9E+09,9E+09,9E+09,9E+09,9E+09,9E+09]];
    CONST robtarget Target_50_2:=[[1267.896290257,-204.087145304,795.115499606],[0.560373641,-0.696206087,0.349493238,-0.281305783],[-1,-2,0,0],[9E+09,9E+09,9E+09,9E+09,9E+09,9E+09]];
    CONST robtarget Target_50_3:=[[1255.043844187,-213.662524168,721.847998286],[0.560373641,-0.696206087,0.349493238,-0.281305783],[-1,-2,0,0],[9E+09,9E+09,9E+09,9E+09,9E+09,9E+09]];
    CONST robtarget Target_50_4:=[[1242.191398117,-223.237903032,648.580496966],[0.560373641,-0.696206087,0.349493238,-0.281305783],[-1,-2,0,0],[9E+09,9E+09,9E+09,9E+09,9E+09,9E+09]];
    CONST robtarget Target_50_5:=[[1229.338952047,-232.813281896,575.312995646],[0.560373641,-0.696206087,0.349493238,-0.281305783],[-1,-2,0,0],[9E+09,9E+09,9E+09,9E+09,9E+09,9E+09]];
    CONST robtarget Target_50_6:=[[1216.486505977,-242.38866076,502.045494326],[0.560373641,-0.696206087,0.349493238,-0.281305783],[-1,-2,0,0],[9E+09,9E+09,9E+09,9E+09,9E+09,9E+09]];
    CONST robtarget Target_50_7:=[[1203.634059907,-251.964039624,428.777993006],[0.560373641,-0.696206087,0.349493238,-0.281305783],[-1,-2,0,0],[9E+09,9E+09,9E+09,9E+09,9E+09,9E+09]];
    CONST robtarget Target_50_8:=[[1190.781613837,-261.539418488,355.510491686],[0.560373641,-0.696206087,0.349493238,-0.281305783],[-1,2,0,0],[9E+09,9E+09,9E+09,9E+09,9E+09,9E+09]];
    CONST robtarget Target_50_9:=[[1177.929167767,-271.114797352,282.242990366],[0.560373641,-0.696206087,0.349493238,-0.281305783],[-1,-2,0,0],[9E+09,9E+09,9E+09,9E+09,9E+09,9E+09]];
    CONST robtarget Target_50_10:=[[1165.076721697,-280.690176216,208.975489046],[0.560373641,-0.696206087,0.349493238,-0.281305783],[-1,-2,0,0],[9E+09,9E+09,9E+09,9E+09,9E+09,9E+09]];
    CONST robtarget Target_60:=[[1443.058680851,-338.903779098,868.383001307],[0.60565287,-0.75246083,0.201621276,-0.1622842],[0,0,0,0],[9E+09,9E+09,9E+09,9E+09,9E+09,9E+09]];
    CONST robtarget Target_60_2:=[[1435.045047672,-352.783798425,795.115500007],[0.60565287,-0.75246083,0.201621276,-0.1622842],[0,0,0,0],[9E+09,9E+09,9E+09,9E+09,9E+09,9E+09]];
    CONST robtarget Target_60_3:=[[1427.031414493,-366.663817752,721.847998707],[0.60565287,-0.75246083,0.201621276,-0.1622842],[0,0,0,0],[9E+09,9E+09,9E+09,9E+09,9E+09,9E+09]];
    CONST robtarget Target_60_4:=[[1419.017781314,-380.543837079,648.580497407],[0.60565287,-0.75246083,0.201621276,-0.1622842],[0,0,0,0],[9E+09,9E+09,9E+09,9E+09,9E+09,9E+09]];
    CONST robtarget Target_60_5:=[[1411.004148135,-394.423856406,575.312996107],[0.60565287,-0.75246083,0.201621276,-0.1622842],[0,0,0,0],[9E+09,9E+09,9E+09,9E+09,9E+09,9E+09]];
    CONST robtarget Target_60_6:=[[1402.990514956,-408.303875733,502.045494807],[0.60565287,-0.75246083,0.201621276,-0.1622842],[0,0,0,0],[9E+09,9E+09,9E+09,9E+09,9E+09,9E+09]];
    CONST robtarget Target_60_7:=[[1394.976881777,-422.18389506,428.777993507],[0.60565287,-0.75246083,0.201621276,-0.1622842],[0,0,0,0],[9E+09,9E+09,9E+09,9E+09,9E+09,9E+09]];
    CONST robtarget Target_60_8:=[[1386.963248598,-436.063914387,355.510492207],[0.60565287,-0.75246083,0.201621276,-0.1622842],[0,0,0,0],[9E+09,9E+09,9E+09,9E+09,9E+09,9E+09]];
    CONST robtarget Target_60_9:=[[1378.949615419,-449.943933714,282.242990907],[0.60565287,-0.75246083,0.201621276,-0.1622842],[0,0,0,0],[9E+09,9E+09,9E+09,9E+09,9E+09,9E+09]];
    CONST robtarget Target_60_10:=[[1370.93598224,-463.823953041,208.975489607],[0.60565287,-0.75246083,0.201621276,-0.1622842],[0,0,0,0],[9E+09,9E+09,9E+09,9E+09,9E+09,9E+09]];
    CONST robtarget Target_20_5:=[[1054.079951383,601.444356528,575.311187629],[0.297972567,-0.370202913,0.685420605,-0.551688994],[0,-1,0,0],[9E+09,9E+09,9E+09,9E+09,9E+09,9E+09]];
    CONST robtarget Target_20_4:=[[1222.069851038,447.825608779,648.580497065],[0.297974422,-0.370202292,0.685418633,-0.55169086],[0,0,0,0],[9E+09,9E+09,9E+09,9E+09,9E+09,9E+09]];
    CONST robtarget Target_70:=[[1284.230996496,544.204446386,1612.651813404],[0.253617413,-0.315094805,0.712437168,-0.573434175],[0,-1,-1,0],[9E+09,9E+09,9E+09,9E+09,9E+09,9E+09]];
    CONST robtarget Target_70_2:=[[936.431880156,489.590660864,590.118183906],[0.297969084,-0.370203288,0.685423834,-0.551686613],[0,-1,0,0],[9E+09,9E+09,9E+09,9E+09,9E+09,9E+09]];
    CONST robtarget Target_70_3:=[[1063.78699175,451.903359442,614.02053489],[0.297969102,-0.370203349,0.68542382,-0.551686579],[0,-1,0,0],[9E+09,9E+09,9E+09,9E+09,9E+09,9E+09]];
    CONST robtarget Target_70_4:=[[922.964386502,533.207464713,620.382968538],[0.297968193,-0.370203343,0.685424653,-0.551686038],[0,-1,0,0],[9E+09,9E+09,9E+09,9E+09,9E+09,9E+09]];
    CONST robtarget Target_70_5:=[[1050.284951926,550.901961563,610.761587013],[0.29797142,-0.370203357,0.685421706,-0.551687949],[0,-1,0,0],[9E+09,9E+09,9E+09,9E+09,9E+09,9E+09]];
    CONST robtarget Target_70_6:=[[1193.597215996,310.429064526,562.397365111],[0.421171477,-0.648741055,-0.281309515,-0.567991714],[0,0,0,0],[9E+09,9E+09,9E+09,9E+09,9E+09,9E+09]];
    CONST robtarget Target_80:=[[1284.230889105,544.204803524,950.074876063],[0.253617391,-0.315095638,0.712437658,-0.573433118],[0,-1,-1,0],[9E+09,9E+09,9E+09,9E+09,9E+09,9E+09]];
    CONST robtarget Target_80_2:=[[1390.564378519,204.430044766,536.36361857],[0.320628157,-0.722452389,-0.366000587,-0.491226731],[0,0,0,0],[9E+09,9E+09,9E+09,9E+09,9E+09,9E+09]];
    CONST robtarget Target_80_3:=[[1369.468422532,217.592102533,538.956083874],[0.320628157,-0.722452389,-0.366000587,-0.491226731],[0,0,0,0],[9E+09,9E+09,9E+09,9E+09,9E+09,9E+09]];
    CONST robtarget Target_80_4:=[[1327.276510559,243.916218067,544.141014483],[0.320628157,-0.722452389,-0.366000587,-0.491226731],[0,0,0,0],[9E+09,9E+09,9E+09,9E+09,9E+09,9E+09]];
    CONST robtarget Target_80_5:=[[1263.9886426,283.402391368,551.918410397],[0.320628157,-0.722452389,-0.366000587,-0.491226731],[0,0,0,0],[9E+09,9E+09,9E+09,9E+09,9E+09,9E+09]];
    CONST robtarget Target_80_6:=[[1200.700774641,322.888564669,559.695806311],[0.320628157,-0.722452389,-0.366000587,-0.491226731],[0,0,0,0],[9E+09,9E+09,9E+09,9E+09,9E+09,9E+09]];
    CONST robtarget Target_90:=[[1245.612941444,477.316882469,950.074675434],[0.253617341,-0.315095893,0.712437846,-0.573432767],[0,-1,-1,0],[9E+09,9E+09,9E+09,9E+09,9E+09,9E+09]];
    CONST robtarget Target_90_2:=[[1398.679661545,215.664462103,560.625108455],[0.221902719,-0.776129388,-0.448013403,-0.384273792],[0,0,0,0],[9E+09,9E+09,9E+09,9E+09,9E+09,9E+09]];
    CONST robtarget Target_90_3:=[[1377.030273168,228.166620806,560.628379067],[0.221902719,-0.776129388,-0.448013403,-0.384273792],[0,0,0,0],[9E+09,9E+09,9E+09,9E+09,9E+09,9E+09]];
    CONST robtarget Target_90_4:=[[1333.731496415,253.170938212,560.634920292],[0.221902719,-0.776129388,-0.448013403,-0.384273792],[0,0,0,0],[9E+09,9E+09,9E+09,9E+09,9E+09,9E+09]];
    CONST robtarget Target_90_5:=[[1268.783331286,290.677414321,560.64473213],[0.221902719,-0.776129388,-0.448013403,-0.384273792],[0,0,0,0],[9E+09,9E+09,9E+09,9E+09,9E+09,9E+09]];
    CONST robtarget Target_90_6:=[[1203.835166157,328.18389043,560.654543968],[0.221902719,-0.776129388,-0.448013403,-0.384273792],[0,0,0,0],[9E+09,9E+09,9E+09,9E+09,9E+09,9E+09]];
    CONST robtarget Target_100:=[[1245.613050994,477.317035369,1586.430900064],[0.253617524,-0.315096302,0.712437895,-0.5734324],[0,-1,-1,0],[9E+09,9E+09,9E+09,9E+09,9E+09,9E+09]];
    CONST robtarget Target_100_2:=[[1413.72309208,244.878612139,588.45862328],[0.109136557,-0.830643309,-0.507852627,-0.200515872],[0,0,0,0],[9E+09,9E+09,9E+09,9E+09,9E+09,9E+09]];
    CONST robtarget Target_100_3:=[[1391.536692169,256.387358205,587.899675204],[0.109136557,-0.830643309,-0.507852627,-0.200515872],[0,0,0,0],[9E+09,9E+09,9E+09,9E+09,9E+09,9E+09]];
    CONST robtarget Target_100_4:=[[1347.163892346,279.404850337,586.781779053],[0.109136557,-0.830643309,-0.507852627,-0.200515872],[0,0,0,0],[9E+09,9E+09,9E+09,9E+09,9E+09,9E+09]];
    CONST robtarget Target_100_5:=[[1280.604692611,313.931088535,585.104934827],[0.109136557,-0.830643309,-0.507852627,-0.200515872],[0,0,0,0],[9E+09,9E+09,9E+09,9E+09,9E+09,9E+09]];
    CONST robtarget Target_100_6:=[[1214.045492876,348.457326733,583.428090601],[0.109136557,-0.830643309,-0.507852627,-0.200515872],[0,0,0,0],[9E+09,9E+09,9E+09,9E+09,9E+09,9E+09]];
    CONST robtarget Target_110:=[[1141.057152561,103.202646089,1559.628873229],[0.355009024,-0.617043491,0.470450565,-0.521442411],[0,-1,-1,0],[9E+09,9E+09,9E+09,9E+09,9E+09,9E+09]];
    CONST robtarget Target_110_2:=[[1432.744350583,280.67669963,599.809032838],[0.014281613,-0.863462424,-0.503591311,-0.02498939],[0,0,0,0],[9E+09,9E+09,9E+09,9E+09,9E+09,9E+09]];
    CONST robtarget Target_110_3:=[[1410.984897443,292.986290984,599.796392664],[0.014281613,-0.863462424,-0.503591311,-0.02498939],[0,0,0,0],[9E+09,9E+09,9E+09,9E+09,9E+09,9E+09]];
    CONST robtarget Target_110_4:=[[1367.465991164,317.605473692,599.771112315],[0.014281613,-0.863462424,-0.503591311,-0.02498939],[0,0,0,0],[9E+09,9E+09,9E+09,9E+09,9E+09,9E+09]];
    CONST robtarget Target_110_5:=[[1302.187631746,354.534247754,599.733191791],[0.014281613,-0.863462424,-0.503591311,-0.02498939],[0,0,0,0],[9E+09,9E+09,9E+09,9E+09,9E+09,9E+09]];
    CONST robtarget Target_110_6:=[[1236.909272328,391.463021816,599.695271267],[0.014281613,-0.863462424,-0.503591311,-0.02498939],[0,0,0,0],[9E+09,9E+09,9E+09,9E+09,9E+09,9E+09]];
    CONST robtarget Target_120:=[[1141.05720731,103.202628921,875.481004344],[0.355008824,-0.617043792,0.470450708,-0.521442063],[0,-2,-1,0],[9E+09,9E+09,9E+09,9E+09,9E+09,9E+09]];
    CONST robtarget Target_120_2:=[[1454.583446133,316.776959216,593.325116018],[0.089334141,0.863795391,0.473534612,-0.147111878],[0,0,0,0],[9E+09,9E+09,9E+09,9E+09,9E+09,9E+09]];
    CONST robtarget Target_120_3:=[[1433.474489698,330.166178336,592.949923358],[0.089334141,0.863795391,0.473534612,-0.147111878],[0,0,0,0],[9E+09,9E+09,9E+09,9E+09,9E+09,9E+09]];
    CONST robtarget Target_120_4:=[[1391.256576826,356.944616577,592.199538039],[0.089334141,0.863795391,0.473534612,-0.147111878],[0,0,0,0],[9E+09,9E+09,9E+09,9E+09,9E+09,9E+09]];
    CONST robtarget Target_120_5:=[[1327.929707519,397.112273939,591.073960061],[0.089334141,0.863795391,0.473534612,-0.147111878],[0,0,0,0],[9E+09,9E+09,9E+09,9E+09,9E+09,9E+09]];
    CONST robtarget Target_120_6:=[[1264.602838212,437.279931301,589.948382083],[0.089334141,0.863795391,0.473534612,-0.147111878],[0,0,0,0],[9E+09,9E+09,9E+09,9E+09,9E+09,9E+09]];
    CONST robtarget Target_130:=[[1219.192151417,-76.031063299,875.479340013],[0.521164558,-0.616172115,0.376632986,-0.454826365],[-1,-2,0,0],[9E+09,9E+09,9E+09,9E+09,9E+09,9E+09]];
    CONST robtarget Target_130_2:=[[1473.378243571,345.524240543,571.152404542],[0.191333663,0.810892673,0.451288014,-0.319661745],[0,0,0,0],[9E+09,9E+09,9E+09,9E+09,9E+09,9E+09]];
    CONST robtarget Target_130_3:=[[1452.022833755,358.510768441,570.607826973],[0.191333663,0.810892673,0.451288014,-0.319661745],[0,0,0,0],[9E+09,9E+09,9E+09,9E+09,9E+09,9E+09]];
    CONST robtarget Target_130_4:=[[1409.312014121,384.483824236,569.518671836],[0.191333663,0.810892673,0.451288014,-0.319661745],[0,0,0,0],[9E+09,9E+09,9E+09,9E+09,9E+09,9E+09]];
    CONST robtarget Target_130_5:=[[1345.245784671,423.443407928,567.884939131],[0.191333663,0.810892673,0.451288014,-0.319661745],[0,0,0,0],[9E+09,9E+09,9E+09,9E+09,9E+09,9E+09]];
    CONST robtarget Target_130_6:=[[1281.179555221,462.40299162,566.251206426],[0.191333663,0.810892673,0.451288014,-0.319661745],[0,0,0,0],[9E+09,9E+09,9E+09,9E+09,9E+09,9E+09]];
    CONST robtarget Target_140:=[[1219.192140749,-76.031140416,1538.266913197],[0.521164325,-0.616172116,0.376633168,-0.454826479],[-1,-2,0,0],[9E+09,9E+09,9E+09,9E+09,9E+09,9E+09]];
    CONST robtarget Target_140_2:=[[1481.249405785,359.103666461,551.10010584],[0.243000339,0.740112555,0.446510357,-0.440241686],[0,0,0,0],[9E+09,9E+09,9E+09,9E+09,9E+09,9E+09]];
    CONST robtarget Target_140_3:=[[1459.377065777,371.182633275,551.936349371],[0.243000339,0.740112555,0.446510357,-0.440241686],[0,0,0,0],[9E+09,9E+09,9E+09,9E+09,9E+09,9E+09]];
    CONST robtarget Target_140_4:=[[1415.63238576,395.340566904,553.608836433],[0.243000339,0.740112555,0.446510357,-0.440241686],[0,0,0,0],[9E+09,9E+09,9E+09,9E+09,9E+09,9E+09]];
    CONST robtarget Target_140_5:=[[1350.015365734,431.577467348,556.117567026],[0.243000339,0.740112555,0.446510357,-0.440241686],[0,0,0,0],[9E+09,9E+09,9E+09,9E+09,9E+09,9E+09]];
    CONST robtarget Target_140_6:=[[1284.398345708,467.814367792,558.626297619],[0.243000339,0.740112555,0.446510357,-0.440241686],[0,0,0,0],[9E+09,9E+09,9E+09,9E+09,9E+09,9E+09]];
    CONST robtarget Target_150:=[[1525.542632187,349.720396937,500],[0.281309515,0.567991714,0.421171477,-0.648741055],[0,0,0,0],[9E+09,9E+09,9E+09,9E+09,9E+09,9E+09]];
    CONST robtarget Target_150_2:=[[1483.370738117,374.068351307,511.344975474],[0.281309515,0.567991714,0.421171477,-0.648741055],[0,0,0,0],[9E+09,9E+09,9E+09,9E+09,9E+09,9E+09]];
    CONST robtarget Target_150_3:=[[1462.284791082,386.242328492,517.017463212],[0.281309515,0.567991714,0.421171477,-0.648741055],[0,0,0,0],[9E+09,9E+09,9E+09,9E+09,9E+09,9E+09]];
    CONST robtarget Target_150_4:=[[1420.112897012,410.590282862,528.362438687],[0.281309515,0.567991714,0.421171477,-0.648741055],[0,0,0,0],[9E+09,9E+09,9E+09,9E+09,9E+09,9E+09]];
    CONST robtarget Target_150_5:=[[1356.855055907,447.112214417,545.379901899],[0.281309515,0.567991714,0.421171477,-0.648741055],[0,0,0,0],[9E+09,9E+09,9E+09,9E+09,9E+09,9E+09]];
    CONST robtarget Target_70_5_2:=[[962.446946449,601.615595456,646.293510977],[0.297970098,-0.370203878,0.685422946,-0.551686772],[0,-1,0,0],[9E+09,9E+09,9E+09,9E+09,9E+09,9E+09]];
    CONST robtarget Target_70_4_2:=[[861.412432414,527.488298524,609.682583811],[0.297966595,-0.370203744,0.685426164,-0.551684756],[0,-1,0,0],[9E+09,9E+09,9E+09,9E+09,9E+09,9E+09]];
    CONST robtarget Target_10_5_2:=[[1380.322671584,628.818480655,575.312996698],[0.181966227,-0.158701032,-0.874817535,0.4199959],[0,0,0,0],[9E+09,9E+09,9E+09,9E+09,9E+09,9E+09]];
    CONST robtarget Target_10_6_2:=[[1371.491810194,642.193425292,502.045495423],[0.216840729,-0.106197101,-0.736305912,0.632104325],[0,0,0,1],[9E+09,9E+09,9E+09,9E+09,9E+09,9E+09]];
    CONST robtarget Target_30_7_2:=[[1087.602745303,236.067470121,428.7779929],[0.706951693,-0.693785733,0.136606578,0.014808877],[0,0,0,0],[9E+09,9E+09,9E+09,9E+09,9E+09,9E+09]];
    CONST robtarget Target_20_5_2:=[[900.353753769,591.307684466,642.382661547],[0.297968237,-0.370204075,0.685424696,-0.551685471],[0,-1,0,0],[9E+09,9E+09,9E+09,9E+09,9E+09,9E+09]];
    CONST robtarget Target_20_6_3:=[[925.071109276,515.981714874,554.541186649],[0.297970412,-0.370202419,0.685422309,-0.551688373],[0,-1,0,0],[9E+09,9E+09,9E+09,9E+09,9E+09,9E+09]];
    CONST robtarget Target_20_7_2:=[[937.807883883,535.37943424,549.43245993],[0.297970812,-0.370202027,0.685421711,-0.551689163],[0,-1,0,0],[9E+09,9E+09,9E+09,9E+09,9E+09,9E+09]];
    CONST robtarget Target_20_8_3:=[[972.6373559,515.287857356,521.51944556],[0.297969697,-0.370201991,0.685423016,-0.551688168],[0,-1,0,0],[9E+09,9E+09,9E+09,9E+09,9E+09,9E+09]];
    CONST robtarget Target_20_5_3:=[[941.074776731,540.716263329,652.696738962],[0.297965059,-0.370204736,0.685427341,-0.551683457],[0,-1,0,0],[9E+09,9E+09,9E+09,9E+09,9E+09,9E+09]];
    CONST robtarget Target_30_5_2:=[[1189.316761479,-6.391062894,509.88575824],[0.70694779,-0.693789733,0.136606313,0.014810271],[-1,1,0,0],[9E+09,9E+09,9E+09,9E+09,9E+09,9E+09]];
    CONST robtarget Target_30_6_2:=[[1153.444867466,52.658841918,509.886694136],[0.706949246,-0.69378823,0.136606481,0.014809606],[-1,1,0,0],[9E+09,9E+09,9E+09,9E+09,9E+09,9E+09]];
    CONST robtarget Target_20_4_3:=[[1003.663994918,573.922606991,647.747369487],[0.29797312,-0.370202923,0.685419869,-0.551689604],[0,-1,0,0],[9E+09,9E+09,9E+09,9E+09,9E+09,9E+09]];
    CONST robtarget Target_20_4_3_2:=[[1012.032977691,653.749023046,640.990678025],[0.297971313,-0.370203209,0.68542137,-0.551688523],[0,-1,-1,0],[9E+09,9E+09,9E+09,9E+09,9E+09,9E+09]];
    CONST robtarget Target_30_8_2:=[[1081.742050215,401.927250903,355.509095199],[0.40329203,-0.501051312,0.59648832,-0.48010916],[0,-1,0,0],[9E+09,9E+09,9E+09,9E+09,9E+09,9E+09]];
    CONST robtarget Target_20_8_4:=[[949.848699503,362.498719256,309.629512326],[0.458422026,-0.428519219,0.423558307,-0.653313773],[0,-2,0,1],[9E+09,9E+09,9E+09,9E+09,9E+09,9E+09]];
    CONST robtarget Target_20_8_4_2:=[[972.884352345,479.17006999,296.088143579],[0.433193331,-0.407475696,0.431831098,-0.678106923],[0,-1,0,1],[9E+09,9E+09,9E+09,9E+09,9E+09,9E+09]];
    CONST robtarget Target_10_5_3:=[[1349.133760372,822.760934177,575.311648729],[0.000012169,-0.000013296,-0.779008718,0.627013091],[0,-1,4,1],[9E+09,9E+09,9E+09,9E+09,9E+09,9E+09]];
    CONST robtarget Target_10_8_2:=[[1353.830016948,668.943727465,355.509347866],[0.219770352,-0.01039516,-0.492164808,0.84223912],[0,-1,0,1],[9E+09,9E+09,9E+09,9E+09,9E+09,9E+09]];
    CONST robtarget Target_40_5_2:=[[1022.367159817,3.127150245,575.310199185],[0.384616337,-0.459230238,0.606484569,-0.522832983],[0,-2,0,0],[9E+09,9E+09,9E+09,9E+09,9E+09,9E+09]];
    CONST robtarget Target_40_5_3:=[[1022.367127059,3.127092663,658.609964479],[0.325650755,-0.412656415,0.670846755,-0.523097409],[0,-1,0,0],[9E+09,9E+09,9E+09,9E+09,9E+09,9E+09]];
    CONST robtarget Target_50_5_2:=[[997.820878166,-386.586813847,575.311672794],[0.560372489,-0.696208325,0.34949231,-0.28130369],[-1,-3,0,0],[9E+09,9E+09,9E+09,9E+09,9E+09,9E+09]];
    CONST robtarget Target_50_5_2_2:=[[1097.199980042,-443.963166282,575.311403035],[0.560372148,-0.696208711,0.349492312,-0.281303412],[-1,-3,0,0],[9E+09,9E+09,9E+09,9E+09,9E+09,9E+09]];
    CONST robtarget Target_60_5_2:=[[1613.347260795,-640.771426545,589.643304631],[0.61141827,-0.765220825,-0.159769892,0.122794013],[-1,0,0,1],[9E+09,9E+09,9E+09,9E+09,9E+09,9E+09]];
    CONST robtarget Target_60_5_3:=[[1654.663171695,-664.625343238,589.64287141],[0.594925066,-0.743934952,-0.240107963,0.187011011],[-1,0,0,1],[9E+09,9E+09,9E+09,9E+09,9E+09,9E+09]];
    CONST robtarget Target_50_6_2:=[[969.464793859,-560.401720905,598.074984018],[0.560371174,-0.696210063,0.34949204,-0.281302345],[-1,-3,0,0],[9E+09,9E+09,9E+09,9E+09,9E+09,9E+09]];
    CONST robtarget Target_50_6_2_2:=[[809.487135382,-468.038734191,598.074764777],[0.560370724,-0.696210307,0.349492257,-0.281302366],[-1,-3,0,0],[9E+09,9E+09,9E+09,9E+09,9E+09,9E+09]];
    CONST robtarget Target_40_6_2:=[[1013.237054504,100.108765216,563.372979398],[0.313577941,-0.38959177,0.674589262,-0.542970032],[0,-1,0,0],[9E+09,9E+09,9E+09,9E+09,9E+09,9E+09]];
    CONST robtarget Target_40_6_2_2:=[[1013.236991894,100.108771544,563.372279499],[0.282401467,-0.276313921,0.674835642,-0.623295183],[0,-1,0,0],[9E+09,9E+09,9E+09,9E+09,9E+09,9E+09]];
    CONST robtarget Target_10_10_2:=[[1327.337503244,709.068148477,135.707989048],[0.180363377,-0.224082776,0.746079989,-0.600516954],[0,0,0,0],[9E+09,9E+09,9E+09,9E+09,9E+09,9E+09]];
    CONST robtarget Target_20_10_2:=[[1128.248378125,509.342439966,135.70798786],[0.297974422,-0.370202292,0.685418633,-0.55169086],[0,0,0,0],[9E+09,9E+09,9E+09,9E+09,9E+09,9E+09]];
    CONST robtarget Target_30_10_2:=[[1008.668858164,249.899069028,62.439208238],[0.377742049,-0.533918067,0.556172687,-0.512751776],[0,-6,4,0],[9E+09,9E+09,9E+09,9E+09,9E+09,9E+09]];
    CONST robtarget Target_40_10_2:=[[1032.907830815,-34.745643496,135.707988167],[0.491980647,-0.611234891,0.482949633,-0.388724329],[-1,-2,0,0],[9E+09,9E+09,9E+09,9E+09,9E+09,9E+09]];
    CONST robtarget Target_60_10_2:=[[1362.922349061,-477.703972368,135.707988307],[0.60565287,-0.75246083,0.201621276,-0.1622842],[0,0,0,0],[9E+09,9E+09,9E+09,9E+09,9E+09,9E+09]];
    CONST robtarget Target_60_10_2_2:=[[1354.908715882,-491.583991695,62.440487007],[0.60565287,-0.75246083,0.201621276,-0.1622842],[0,0,0,0],[9E+09,9E+09,9E+09,9E+09,9E+09,9E+09]];
    CONST robtarget Target_50_10_2_2:=[[1139.371829557,-299.840933944,62.440486406],[0.560373641,-0.696206087,0.349493238,-0.281305783],[-1,-2,0,0],[9E+09,9E+09,9E+09,9E+09,9E+09,9E+09]];
    CONST robtarget Target_40_10_2_2:=[[1017.315207922,-38.452847816,62.440486862],[0.491980647,-0.611234891,0.482949633,-0.388724329],[-1,-2,0,0],[9E+09,9E+09,9E+09,9E+09,9E+09,9E+09]];
    CONST robtarget Target_30_10_2_2:=[[1008.669104053,249.899010996,62.44048628],[0.403294899,-0.501052053,0.596485774,-0.480109139],[0,-2,0,0],[9E+09,9E+09,9E+09,9E+09,9E+09,9E+09]];
    CONST robtarget Target_20_10_2_2:=[[1114.845310566,518.130558707,62.440486545],[0.297974422,-0.370202292,0.685418633,-0.55169086],[0,0,0,0],[9E+09,9E+09,9E+09,9E+09,9E+09,9E+09]];
    CONST robtarget Target_10_10_2_2:=[[1344.459653043,722.563356422,62.440002939],[0.180362226,-0.224082488,0.746081324,-0.600515749],[0,-1,0,0],[9E+09,9E+09,9E+09,9E+09,9E+09,9E+09]];
    CONST robtarget Target_50_10_2:=[[1152.224275627,-290.26555508,135.707987726],[0.560373641,-0.696206087,0.349493238,-0.281305783],[-1,-2,0,0],[9E+09,9E+09,9E+09,9E+09,9E+09,9E+09]];
    CONST robtarget Target_60_5_4:=[[1172.965926879,-443.200347487,713.204222749],[0.489405782,-0.816709315,0.236661397,-0.193543946],[-1,1,0,0],[9E+09,9E+09,9E+09,9E+09,9E+09,9E+09]];
    CONST robtarget Target_60_5_5:=[[1084.320997093,-458.967006799,739.46130536],[0.489404876,-0.816709915,0.236661427,-0.193543669],[-1,1,0,0],[9E+09,9E+09,9E+09,9E+09,9E+09,9E+09]];
    CONST robtarget Target_40_7_2:=[[1080.723946367,-11.51415719,428.775060534],[0.326528534,-0.311874116,0.640161959,-0.621535452],[0,-1,0,0],[9E+09,9E+09,9E+09,9E+09,9E+09,9E+09]];
    CONST robtarget Target_50_7_2:=[[1011.225965863,-427.061011806,478.873678061],[0.560371664,-0.696211257,0.349490163,-0.281300746],[-1,-3,0,0],[9E+09,9E+09,9E+09,9E+09,9E+09,9E+09]];
    CONST robtarget Target_50_8_2:=[[1143.051951896,-490.181950167,325.706026838],[0.769454079,-0.326774391,0.467925322,0.286713815],[-1,1,1,1],[9E+09,9E+09,9E+09,9E+09,9E+09,9E+09]];
    CONST robtarget Target_50_8_3:=[[1002.836973024,-409.228984788,325.703744713],[0.757261174,-0.173863831,0.56068758,0.286280141],[-1,1,1,1],[9E+09,9E+09,9E+09,9E+09,9E+09,9E+09]];
    CONST robtarget Target_60_8_2:=[[1217.001042404,-418.462464534,244.095724308],[0.79769968,-0.266578995,0.434139659,0.322697407],[-1,1,1,1],[9E+09,9E+09,9E+09,9E+09,9E+09,9E+09]];
    CONST robtarget Target_60_8_3:=[[1247.415991324,-365.782295085,246.341111536],[0.86279693,-0.278736127,0.333391019,0.258337101],[-1,1,1,1],[9E+09,9E+09,9E+09,9E+09,9E+09,9E+09]];
    CONST robtarget Target_60_8_4:=[[1219.426116168,-414.263078329,246.336374316],[0.865191582,-0.310960843,0.31358895,0.237505478],[-1,1,1,1],[9E+09,9E+09,9E+09,9E+09,9E+09,9E+09]];
	CONST robtarget Target_160:=[[1175.200656563,474.230762615,157.162932039],[0.18035962,-0.224080292,0.746083038,-0.600515221],[0,-1,0,0],[9E+09,9E+09,9E+09,9E+09,9E+09,9E+09]];
    CONST robtarget Target_170:=[[1325.529881312,-387.193695954,64.002538181],[0.53756845,-0.646192069,0.438010474,-0.318751935],[-1,-2,0,0],[9E+09,9E+09,9E+09,9E+09,9E+09,9E+09]];
PROC Path_10()
         ColorIndex2:=1;
         Set do2;
         WaitTime 1;
        MoveL Target_70,v1000,z100,tool0\WObj:=wobj0;
        MoveL Target_80,v1000,z100,tool0\WObj:=wobj0;
        MoveL Target_90,v1000,z100,tool0\WObj:=wobj0;
        MoveL Target_100,v1000,z100,tool0\WObj:=wobj0;
        MoveL Target_110,v1000,z100,tool0\WObj:=wobj0;
        MoveL Target_120,v1000,z100,tool0\WObj:=wobj0;
        MoveL Target_130,v1000,z100,tool0\WObj:=wobj0;
        MoveL Target_140,v1000,z100,tool0\WObj:=wobj0;
        MoveL Target_10,v500,fine,tool0\WObj:=wobj0;
        MoveL Target_20,v500,fine,tool0\WObj:=wobj0;
        MoveL Target_30,v500,fine,tool0\WObj:=wobj0;
        MoveL Target_40,v500,fine,tool0\WObj:=wobj0;
        MoveL Target_50,v500,fine,tool0\WObj:=wobj0;
        MoveL Target_60,v500,fine,tool0\WObj:=wobj0;
        MoveL Target_60_2,v500,fine,tool0\WObj:=wobj0;
        MoveL Target_50_2,v500,fine,tool0\WObj:=wobj0;
        MoveL Target_40_2,v500,fine,tool0\WObj:=wobj0;
        MoveL Target_30_2,v500,fine,tool0\WObj:=wobj0;
        MoveL Target_20_2,v500,fine,tool0\WObj:=wobj0;
        MoveL Target_10_2,v500,fine,tool0\WObj:=wobj0;
        MoveL Target_10_3,v500,fine,tool0\WObj:=wobj0;
	    MoveL Target_20_3,v500,fine,tool0\WObj:=wobj0;
	    MoveL Target_30_3,v500,fine,tool0\WObj:=wobj0;
	    MoveL Target_40_3,v500,fine,tool0\WObj:=wobj0;
        MoveL Target_50_3,v500,fine,tool0\WObj:=wobj0;
        MoveL Target_60_3,v500,fine,tool0\WObj:=wobj0;
        MoveL Target_60_4,v500,fine,tool0\WObj:=wobj0;
        MoveL Target_50_4,v500,fine,tool0\WObj:=wobj0;
        MoveL Target_40_4,v500,fine,tool0\WObj:=wobj0;
        MoveL Target_30_4,v500,fine,tool0\WObj:=wobj0;
        MoveL Target_20_4,v500,fine,tool0\WObj:=wobj0;
        MoveL Target_20_4_3,v500,fine,tool0\WObj:=wobj0;
        MoveL Target_20_4_3_2,v500,fine,tool0\WObj:=wobj0;
        MoveL Target_20_4,v500,fine,tool0\WObj:=wobj0;
        MoveL Target_10_4,v500,fine,tool0\WObj:=wobj0;
        MoveL Target_10_5,v500,fine,tool0\WObj:=wobj0;
        MoveL Target_10_5_3,v500,fine,tool0\WObj:=wobj0;
        MoveL Target_10_5,v500,fine,tool0\WObj:=wobj0;
        MoveL Target_10_5_2,v1000,z100,tool0\WObj:=wobj0;
        MoveL Target_20_5,v1000,z100,tool0\WObj:=wobj0;
        MoveL Target_20_5_2,v1000,z100,tool0\WObj:=wobj0;
        MoveL Target_20_5_3,v1000,z100,tool0\WObj:=wobj0;
        MoveL Target_30_5,v500,fine,tool0\WObj:=wobj0;
        MoveL Target_30_5_2,v1000,z100,tool0\WObj:=wobj0;
        MoveL Target_30_5,v500,fine,tool0\WObj:=wobj0;
        MoveL Target_40_5,v500,fine,tool0\WObj:=wobj0;
        MoveL Target_40_5_2,v500,fine,tool0\WObj:=wobj0;
        MoveL Target_40_5_3,v500,fine,tool0\WObj:=wobj0;
        MoveL Target_40_5,v500,fine,tool0\WObj:=wobj0;
        MoveL Target_50_5,v500,fine,tool0\WObj:=wobj0;
        MoveL Target_50_5_2,v500,fine,tool0\WObj:=wobj0;
        MoveL Target_50_5_2_2,v500,fine,tool0\WObj:=wobj0;
        MoveL Target_50_5,v500,fine,tool0\WObj:=wobj0;
        MoveL Target_60_5,v500,fine,tool0\WObj:=wobj0;
        MoveL Target_60_5_2,v500,fine,tool0\WObj:=wobj0;
        MoveL Target_60_5_3,v500,fine,tool0\WObj:=wobj0;
        MoveL Target_60_5_4,v500,fine,tool0\WObj:=wobj0;
        MoveL Target_60_5_5,v500,fine,tool0\WObj:=wobj0;
        MoveL Target_60_5,v500,fine,tool0\WObj:=wobj0;
        MoveL Target_60_6,v500,fine,tool0\WObj:=wobj0;
        MoveL Target_50_6,v500,fine,tool0\WObj:=wobj0;
        MoveL Target_50_6_2,v500,fine,tool0\WObj:=wobj0;
        MoveL Target_50_6_2_2,v500,fine,tool0\WObj:=wobj0;
        MoveL Target_40_6,v500,fine,tool0\WObj:=wobj0;
        MoveL Target_40_6_2,v500,fine,tool0\WObj:=wobj0;
        MoveL Target_40_6_2_2,v500,fine,tool0\WObj:=wobj0;
        MoveL Target_40_6,v500,fine,tool0\WObj:=wobj0;
        MoveL Target_30_6,v500,fine,tool0\WObj:=wobj0;
        MoveL Target_30_6_2,v1000,z100,tool0\WObj:=wobj0;
        MoveL Target_20_6_3,v500,fine,tool0\WObj:=wobj0;
        MoveL Target_20_6,v500,fine,tool0\WObj:=wobj0;
        MoveL Target_10_6_2,v1000,z100,tool0\WObj:=wobj0;
        MoveL Target_10_6,v500,fine,tool0\WObj:=wobj0;
        MoveL Target_10_7,v500,fine,tool0\WObj:=wobj0;
        MoveL Target_20_7,v500,fine,tool0\WObj:=wobj0;
        MoveL Target_20_7_2,v500,fine,tool0\WObj:=wobj0;
        MoveL Target_30_7,v500,fine,tool0\WObj:=wobj0;
        MoveL Target_30_7_2,v1000,z100,tool0\WObj:=wobj0;
        MoveL Target_40_7,v500,fine,tool0\WObj:=wobj0;
        MoveL Target_40_7_2,v500,fine,tool0\WObj:=wobj0;
        MoveL Target_40_7,v500,fine,tool0\WObj:=wobj0;
        MoveL Target_50_7,v500,fine,tool0\WObj:=wobj0;
        MoveL Target_50_7_2,v500,fine,tool0\WObj:=wobj0;
        MoveL Target_50_7,v500,fine,tool0\WObj:=wobj0;
        MoveL Target_60_7,v500,fine,tool0\WObj:=wobj0;
        MoveL Target_60_8,v500,fine,tool0\WObj:=wobj0;
        MoveL Target_60_8_2,v500,fine,tool0\WObj:=wobj0;
        MoveL Target_60_8_3,v500,fine,tool0\WObj:=wobj0;
        MoveL Target_60_8_4,v500,fine,tool0\WObj:=wobj0;
        MoveL Target_60_8,v500,fine,tool0\WObj:=wobj0;
        MoveL Target_50_8,v500,fine,tool0\WObj:=wobj0;
        MoveL Target_50_8_2,v500,fine,tool0\WObj:=wobj0;
        MoveL Target_50_8_3,v500,fine,tool0\WObj:=wobj0;
        MoveL Target_50_8,v500,fine,tool0\WObj:=wobj0;
        MoveL Target_40_8,v500,fine,tool0\WObj:=wobj0;
        MoveL Target_30_8,v500,fine,tool0\WObj:=wobj0;
        MoveL Target_30_8_2,v500,fine,tool0\WObj:=wobj0;
        MoveL Target_20_8_3,v500,fine,tool0\WObj:=wobj0;
        MoveL Target_30_8_2,v500,fine,tool0\WObj:=wobj0;
        MoveL Target_20_8,v500,fine,tool0\WObj:=wobj0;
        MoveL Target_20_8_4,v500,fine,tool0\WObj:=wobj0;
        MoveL Target_20_8_4_2,v500,fine,tool0\WObj:=wobj0;
        MoveL Target_20_8,v500,fine,tool0\WObj:=wobj0;
        MoveL Target_10_8,v500,fine,tool0\WObj:=wobj0;
        MoveL Target_10_8_2,v500,fine,tool0\WObj:=wobj0;
        MoveL Target_10_8,v500,fine,tool0\WObj:=wobj0;
        MoveL Target_10_9,v500,fine,tool0\WObj:=wobj0;
        MoveL Target_20_9,v500,fine,tool0\WObj:=wobj0;
        MoveL Target_30_9,v500,fine,tool0\WObj:=wobj0;
        MoveL Target_40_9,v500,fine,tool0\WObj:=wobj0;
        MoveL Target_50_9,v500,fine,tool0\WObj:=wobj0;
        MoveL Target_60_9,v500,fine,tool0\WObj:=wobj0;
		MoveL Target_60_10,v500,fine,tool0\WObj:=wobj0;
		MoveL Target_50_10,v500,fine,tool0\WObj:=wobj0;
		MoveL Target_40_10,v500,fine,tool0\WObj:=wobj0;
		MoveL Target_30_10,v500,fine,tool0\WObj:=wobj0;
		MoveL Target_20_10,v500,fine,tool0\WObj:=wobj0;
		MoveL Target_10_10,v500,fine,tool0\WObj:=wobj0;
        MoveL Target_10_10_2,v1000,z100,tool0\WObj:=wobj0;
        MoveL Target_20_10_2,v1000,z100,tool0\WObj:=wobj0;
        MoveL Target_30_10_2,v1000,z100,tool0\WObj:=wobj0;
        MoveL Target_40_10_2,v1000,z100,tool0\WObj:=wobj0;
        MoveL Target_50_10_2,v1000,z100,tool0\WObj:=wobj0;
        MoveL Target_60_10_2,v1000,z100,tool0\WObj:=wobj0;
        MoveL Target_60_10_2_2,v1000,z100,tool0\WObj:=wobj0;
        MoveL Target_50_10_2_2,v1000,z100,tool0\WObj:=wobj0;
        MoveL Target_40_10_2_2,v1000,z100,tool0\WObj:=wobj0;
        MoveL Target_30_10_2_2,v1000,z100,tool0\WObj:=wobj0;
        MoveL Target_20_10_2_2,v1000,z100,tool0\WObj:=wobj0;
        MoveL Target_10_10_2_2,v1000,fine,tool0\WObj:=wobj0;
        MoveL Target_160,v1000,z100,tool0\WObj:=wobj0;
        MoveL Target_170,v1000,fine,tool0\WObj:=wobj0;
        WaitTime 1;
        Reset do2;
    ENDPROC

PROC mai()
     ColorIndex2:=1;
     Set do2;
     WaitTime 1;
    Path_10;



ENDPROC
ENDMODULE

